5030.07 BOOL  ; DROP GUARD FORWARD
5030.08 BOOL  ; EXCHANGE CONVEYOR CW
5030.09 BOOL  ; EXCHANGE CONVEYOR CCW
5030.12 BOOL  ; PALLETIZING CONVEYOR
5030.13 BOOL  ; STACKING CONVEYOR
5040.00 BOOL  ; POSITIONING 1 BACKWARD
5040.01 BOOL  ; POSITIONING 1 FORWARD
5040.02 BOOL  ; LIFTER DOWNWARD
5040.03 BOOL  ; LIFTER UPWARD
5040.04 BOOL  ; POSITIONING 2 BACKWARD
5040.05 BOOL  ; POSITIONING 2 FORWARD
5040.06 BOOL  ; DROP GUARD BACKWARD
5040.07 BOOL  ; DROP GUARD FORWARD
5040.08 BOOL  ; EXCHANGE CONVEYOR CW
5040.09 BOOL  ; EXCHANGE CONVEYOR CCW
5040.10 BOOL  ; Writing of ID3
5040.11 BOOL  ; Writing of ID4
5040.12 BOOL  ; PALLETIZING CONVEYOR
5040.13 BOOL  ; STACKING CONVEYOR
5040.14 BOOL  ; CONVEYOR STOP
5043.00 BOOL  ; STOPPER DOWNWARD SIGNAL
5043.01 BOOL  ; Writing signal of ID3
5043.02 BOOL  ; Writing signal of ID4
5043.03 BOOL  ; STACKING CONVEYOR START SIGNAL
5043.05 BOOL  ; PALLETIZING CONVEYOR STOP SIGNAL
5043.06 BOOL  ; ﾚｰﾝ2段積み部ｺﾝﾍﾞｱ停止信号
5045.00 BOOL  ; 19ST_HOME POSITION
5045.01 BOOL  ; 19ST_CYCLE RUNNING
5052.03 BOOL  ; STACKING CONVEYOR START SIGNAL
5052.06 BOOL  ; STACKING CONVEYOR STOP SIGNAL
5052.07 BOOL  ; STACKING IMPROPRIETY
5052.08 BOOL  ; Downward confirmation when product number is switched
5052.10 BOOL  ; Disbursement completion of fraction workpiece
5053.00 BOOL  ; 20ST_1CY START PB on
5053.01 BOOL  ; 20ST_1CY RUN
5053.02 BOOL  ; 20ST_INDIV STEP START
5053.03 BOOL  ; 20ST_UNIT HOME POSITION PB
5053.04 BOOL  ; 20ST_UNIT HOME POSITION PB PLUSE
5054.00 BOOL  ; 20ST_CONDITION OF START(AUTO)
5054.01 BOOL  ; 20ST_CONDITION OF START(INDIV)
5054.04 BOOL  ; 20ST_CONDITION OF CYCLE START
5054.08 BOOL  ; 20ST_START RESET
5054.09 BOOL  ; 20ST_STEP UP ENABLE
5055.00 BOOL  ; 20ST_CYCLE RUNNING
5055.01 BOOL  ; 20ST_CYCLE RUNNING PLUSE
5055.02 BOOL  ; 20ST_STEP UP ENABLE
5055.03 BOOL  ; UNLOADING UNIT START
5055.04 BOOL  ; STACKING START
5055.05 BOOL  ; UNLOADING  START OF STACKING CONTAINER
5055.06 BOOL  ; UNLOADING PALLET CONVEYOR
5055.15 BOOL  ; 20ST_CYCLE COMPLETE
5056.08 BOOL  ; UNLOADING CONVEYOR 1
5056.12 BOOL  ; UNLOADING CONVEYOR 2
5056.13 BOOL  ; UNLOADING UNIT STOP
5057.00 BOOL  ; STACKING HOOK BACKWARD END
5057.01 BOOL  ; STACKING HOOK FORWARD END
5057.08 BOOL  ; STACKING LIFTER DOWNWARD END
5057.09 BOOL  ; STACKING LIFTER UPWARD END
5057.10 BOOL  ; STACKING LIFTER INTERMEDIATE POSITION
5080.00 BOOL  ; STACKING HOOK BACKWARD
5080.01 BOOL  ; STACKING HOOK FORWARD
5080.02 BOOL  ; STACKING LIFTER DOWNWARD
5080.03 BOOL  ; STACKING LIFTER UPWARD
5080.04 BOOL  ; STACKING CONVEYOR
5080.06 BOOL  ; STACKING STOPPER DOWNWARD
5080.07 BOOL  ; STACKING STOPPER UPWARD
5080.08 BOOL  ; UNLOADING CONVEYOR 1
5080.10 BOOL  ; UNLOADING ESCAPE UPWARD
5080.11 BOOL  ; UNLOADING ESCAPE DOWNWARD
5080.12 BOOL  ; UNLOADING CONVEYOR 2
5080.14 BOOL  ; UNLOADING STOPPER DOWNWARD
5080.15 BOOL  ; UNLOADING STOPPER UPWARD
5090.00 BOOL  ; STACKING HOOK BACKWARD
5090.01 BOOL  ; STACKING HOOK FORWARD
5090.02 BOOL  ; STACKING LIFTER DOWNWARD
5090.03 BOOL  ; STACKING LIFTER UPWARD
5090.04 BOOL  ; STACKING CONVEYOR
5090.05 BOOL  ; CONVEYOR STOP
5090.06 BOOL  ; STACKING STOPPER DOWNWARD
5090.07 BOOL  ; STACKING STOPPER UPWARD
5090.08 BOOL  ; UNLOADING CONVEYOR 1
5090.10 BOOL  ; UNLOADING ESCAPE UPWARD
5090.11 BOOL  ; UNLOADING ESCAPE DOWNWARD
5090.12 BOOL  ; UNLOADING CONVEYOR 2
5090.14 BOOL  ; UNLOADING STOPPER DOWNWARD
5090.15 BOOL  ; UNLOADING STOPPER UPWARD
5093.06 BOOL  ; STACKING CONVEYOR STOP SIGNAL
5093.07 BOOL  ; Container discharge completion
5093.08 BOOL  ; Stacking containers cannot be exchanged
5095.00 BOOL  ; 20ST_HOME POSITION
5095.01 BOOL  ; 20ST_CYCLE RUNNING
5100.00 BOOL  ; PB_Master On
5100.01 BOOL  ; PB_HOME_POS_RE
5100.02 BOOL  ; MASTER ON CONFIRM
5100.03 BOOL  ; PRO_START
5100.04 BOOL  ; HOME_POST_RE_COND
5100.05 BOOL  ; STEP_STOP_COND
5100.06 BOOL  ; MOMENT_STOP_COND
5100.07 BOOL  ; INTERRUPT_SKIP_COND
5100.08 BOOL  ; SS_PRP_INTLK
5100.09 BOOL  ; AIR_SC_CONF
5100.10 BOOL  ; SS_AUTO_IND
5100.11 BOOL  ; TEACHING ON_OFF
5100.12 BOOL  ; PL_AUTO_RUN
5100.13 BOOL  ; PB_FLT RESET
5100.14 BOOL  ; N_E_STOP
5100.15 BOOL  ; N_AUTO_STOP
5101.00 BOOL  ; STOP_COND
5101.01 BOOL  ; ENERGI_SAVING
5101.02 BOOL  ; ENERGI_SAVING_REL
5110.01 BOOL  ; EX_RB_RUNNING
5110.02 BOOL  ; EX_RB_FLT
5110.03 BOOL  ; EX_RB_SERVO_ON
5110.04 BOOL  ; EX_RB_INITIAL_COMPL
5110.05 BOOL  ; EX_RB_AUTO_MODE
5110.06 BOOL  ; EX_RB_OUTSIDE_MODE
5110.07 BOOL  ; EX_RB_BAT_WARNING
5110.08 BOOL  ; EX_RB_WARNING
5110.11 BOOL  ; EX_RB_HOME_POS
5110.14 BOOL  ; EX_COMMAND_TRTMT_COMPL
5110.15 BOOL  ; EX_RB_STATUS_ODD_PARITY
5111.00 BOOL  ; EX_RB_HOME_POS
5111.03 BOOL  ; EX_RB_MOTION_OK
5111.04 BOOL  ; EX_RB_MOTION_NG
5111.06 BOOL  ; EX_RB_SENSOR_CHK_NG
5111.07 BOOL  ; EX_RB_HAND_REP_NG
5111.08 BOOL  ; EX_RB_VISUAL NG
5130.00 BOOL  ; SIG_OFF_COMF
5130.01 BOOL  ; FLT_CODE
5130.02 BOOL  ; COMMAND_FIN
5130.03 BOOL  ; COMMAND_COMP
5130.05 BOOL  ; DATA_AREA1_BIT_EVEN
5130.06 BOOL  ; DATA_AREA2_BIT_EVEN
5130.07 BOOL  ; COMMAND_AREA_BIT_EVEN
5130.10 BOOL  ; DATA_BIT_SUM_ODD
5130.11 BOOL  ; COMMAND_TRTMT_COMPL
5130.12 BOOL  ; RB_FAULT_CLEAR_TIMING
5200.00 BOOL  ; RB_master On Condition
5200.01 BOOL  ; MSTR_ON_AIR_SC_CONF
5200.02 BOOL  ; Master On Confirm
5200.03 BOOL  ; RB_MSTR_ON_1_SCAN
5200.04 BOOL  ; MODE_CHANGE
5200.05 BOOL  ; MODE_CHANGE_COMPL
5200.06 BOOL  ; RB_HOME_POS_PB_ON
5200.07 BOOL  ; RB_HOME_POS_MOTION
5200.08 BOOL  ; RB_HOME_POS_NO_MOTION
5200.09 BOOL  ; RB_HOME_POS_COND_CONFIRM
5200.10 BOOL  ; RB_HOME_POS_PRO_START
5200.11 BOOL  ; PRO_START_RESET
5200.12 BOOL  ; RB_MSTR_ON_COMP_CLEAR_1SCAN
5200.13 BOOL  ; RB_MSTR_ON_COMP_COND
5200.14 BOOL  ; RB_MSTR_ON_COMPL
5200.15 BOOL  ; PL_RB_MSTR_ON
5201.00 BOOL  ; RB_HOME_POS_1SCAN
5201.01 BOOL  ; RB_HOME_POS_1SCAN_MEMORY
5201.02 BOOL  ; RB_HOME_POS
5201.03 BOOL  ; PL_RB_HOME_POS_RE
5201.05 BOOL  ; ENERGY_SAVING_RECEPTION
5201.06 BOOL  ; RB_PRO_START_RESET_CON
5201.07 BOOL  ; ENERGY_SAVING_REL_RECEPTION_CON
5201.09 BOOL  ; ENERGY_SAVING_REL_RECEPTION
5201.10 BOOL  ; STOP
5250.00 BOOL  ; RB_OUTSIDE_START
5250.01 BOOL  ; STROBE_SIGNAL
5250.02 BOOL  ; RB_PROSTART
5250.03 BOOL  ; RB_PRO_START_RESET
5250.04 BOOL  ; RB_RUNNING_CONFIRM
5250.05 BOOL  ; RB_MOVE_OK
5250.06 BOOL  ; RB_MOVE_NG
5400.00 BOOL  ; PL_RB_MASTER ON
5400.01 BOOL  ; PL_RB_HOME POST
5400.02 BOOL  ; CR_RB STOP
5400.03 BOOL  ; RB_FAULT
5400.04 BOOL  ; RB_BAT OFF WARNING
5400.05 BOOL  ; RB WARNING FAULT
5400.06 BOOL  ; SENSOR CHECK NG
5400.07 BOOL  ; HAND REP NG
5400.08 BOOL  ; VISION NG
5400.10 BOOL  ; RB_HOME POST
5400.11 BOOL  ; RB_MOTION OK COMPLETE
5400.12 BOOL  ; RB_MOTION NG COMPLETE
5400.13 BOOL  ; RB SERVO ON
5400.14 BOOL  ; RB_MASTER ON
5600.00 BOOL  ; Task Error Flag
5600.02 BOOL  ; Automatic Mode Flag
5600.03 BOOL  ; Manual Mode Flag
5600.04 BOOL  ; Program Execution Flag
5600.05 BOOL  ; $?St$Bk?_#[18] / Program Execution / Completed Flag$?St$Bk?_#[18]
5600.06 BOOL  ; Optional Input Standby
5600.07 BOOL  ; M Code Reset Standby
5600.08 BOOL  ; M Strobe
5600.09 BOOL  ; Cycle Start Received
5600.13 BOOL  ; Teaching Completed
5600.14 BOOL  ; Teaching Error
5600.15 BOOL  ; Teaching Address Over
5601.00 BOOL  ; Reference Origin
5601.01 BOOL  ; Busy Flag
5601.02 BOOL  ; Servo-lock ON
5601.03 BOOL  ; No Origin Flag
5601.04 BOOL  ; Axis Operating
5601.05 BOOL  ; Positioning Completed
5601.06 BOOL  ; Error Counter Warning
5601.07 BOOL  ; Alarm Input
5602.00 BOOL  ; Servo Lock
5602.01 BOOL  ; Servo Realise
5602.02 BOOL  ; Servo Origin
5604.00 BOOL  ; MC_AutoMan
5605.00 BOOL  ; Servo Motion Start Condition
5605.01 BOOL  ; Servo Motion Start
5605.02 BOOL  ; MC_Read Prog
5605.03 BOOL  ; Servo Motion Start Prog
5605.04 BOOL  ; Servo Motion Moving
5605.05 BOOL  ; Servo Motion Complete
5605.15 BOOL  ; Motion Complete
5610.00 BOOL  ; Servo Forward Position
5610.01 BOOL  ; Servo Backward Position
5650.01 BOOL  ; X AXIS TEACHING &JOG SCREEN
5650.03 BOOL  ; MASTER SWITCH ON TRIGGER
5650.04 BOOL  ; MASTER SWITCH OFF TRIGGER
5650.11 BOOL  ; X AXIS SETTING SCREEN
5651.00 BOOL  ; THE TEACHING IS ACCEPTABLE
5651.01 BOOL  ; TRANSFER ADVANCEMENT EDGE TETI COMPLETION
5651.02 BOOL  ; TRANSFER ADVANCEMENT EDGE TETI INSIDE
5651.04 BOOL  ; TRANSFER ADVANCEMENT SPEED TETI INSIDE
5651.05 BOOL  ; TRANSFER RETREAT SPEED TETI COMPLETION
5651.08 BOOL  ; FLASH MEMORY PRESERVATION TIMING
5651.09 BOOL  ; FRATSUSSHUMEMORI PRESERVATION COMPLETION
5651.10 BOOL  ; THE FLASH MEMORY IS BEING PRESERVED
5651.14 BOOL  ; TRANSFER POSITIONAL DATA READING COMPLETION
5651.15 BOOL  ; TRANSFER POSITIONAL DATA IS BEING READ
5652.00 BOOL  ; FORWARDING PERMISSION
5652.01 BOOL  ; MEMORY DRIVING END
5665.01 BOOL  ; TRANSFER ADVANCEMENT EDGE POSITION
5665.02 BOOL  ; TRANSFER ORIGINAL POSITION
5665.05 BOOL  ; TRANSFER FIXED POSITIONAL CONFIRMATION
6010.04 BOOL  ; During automatic operation from the previous process
6100 CHANNEL  ; AUTO RUNNING MACHINE
6100.01 BOOL  ; AUTO RUNNING OF MACHINE No.1
6100.02 BOOL  ; AUTO RUNNING OF MACHINE No.2
6100.03 BOOL  ; AUTO RUNNING OF MACHINE No.3
6100.04 BOOL  ; AUTO RUNNING OF MACHINE No.4
6100.05 BOOL  ; AUTO RUNNING OF MACHINE No.5
6100.06 BOOL  ; AUTO RUNNING OF MACHINE No.6
6100.07 BOOL  ; AUTO RUNNING OF MACHINE No.7
6100.08 BOOL  ; AUTO RUNNING OF MACHINE No.8
6100.09 BOOL  ; AUTO RUNNING OF MACHINE No.9
6100.10 BOOL  ; AUTO RUNNING OF MACHINE No.10
6100.11 BOOL  ; AUTO RUNNING OF MACHINE No.11
6101 CHANNEL  ; FAULT STOP MACHINE
6101.01 BOOL  ; FAULT STOP OF MACHINE No.1
6101.02 BOOL  ; FAULT STOP OF MACHINE No.2
6101.03 BOOL  ; FAULT STOP OF MACHINE No.3
6101.04 BOOL  ; FAULT STOP OF MACHINE No.4
6101.05 BOOL  ; FAULT STOP OF MACHINE No.5
6101.06 BOOL  ; FAULT STOP OF MACHINE No.6
6101.07 BOOL  ; FAULT STOP OF MACHINE No.7
6101.08 BOOL  ; FAULT STOP OF MACHINE No.8
6101.09 BOOL  ; FAULT STOP OF MACHINE No.9
6101.10 BOOL  ; FAULT STOP OF MACHINE No.10
6101.11 BOOL  ; FAULT STOP OF MACHINE No.11
6102.00 BOOL  ; ALL MACHINE OPERATING
6102.01 BOOL  ; FAULT STOP SIGNAL
6102.02 BOOL  ; DATA MEMORY
6102.03 BOOL  ; ALL MACHINE OPERATING MEMORY
6102.11 BOOL  ; PERIODICAL STOP
6102.12 BOOL  ; FAULT STOP
6102.13 BOOL  ; AUTO RUNNING STOP
6140.00 BOOL  ; CHECK BEARING NEW SENSOR
6140.01 BOOL  ; NO BEARING
6140.07 BOOL  ; KZ COLLECTING NG 291222
6142.07 BOOL  ; XXXXXX
6143.00 BOOL  ; -
6143.03 BOOL  ; Bug fix 20151125
6143.04 BOOL  ; For adjustment when there is no ID information from the previous process
6143.06 BOOL  ; Addition of finishing correction circuit
6143.07 BOOL  ; Measuring unit correction circuit
6143.09 BOOL  ; Shirai correction after 20150803
6143.10 BOOL  ; 山本修正
6143.12 BOOL  ; NO ID
6143.13 BOOL  ; Impulse measurement complete
6143.15 BOOL  ; TEMPORARY CONTACT FOR ADJUSTMENT ON
A343.13 BOOL  ; Flag when file memory operation is being executed
A343.15 BOOL  ; Memory card confirmation flag
A351 CHANNEL  ; Clock data and second
A352 CHANNEL  ; Clock data day and time
A353 CHANNEL  ; The moon clock data every year
A401.06 BOOL  ; FALS FAULT FLAG(STOP)
A402.02 BOOL  ; HIGH EFFICIENT I/O SETTING FAULT
A402.03 BOOL  ; CPU HIGH EFFICIENT I/O SETTING FAULT
A402.05 BOOL  ; SYSBUS FAULT
A402.06 BOOL  ; HIGH EFFICIENT I/O FAULT
A402.07 BOOL  ; CPU HIGH EFFICIENT I/O FAULT
A402.08 BOOL  ; INNER BOARD FAULT
A402.10 BOOL  ; FAULT IN PC SYSTEM CONSTRUCTION
A402.12 BOOL  ; FAULT IN BASIC I/O UNIT
A402.13 BOOL  ; FAULT IN INTERRUPTION TASK
A410.06 BOOL  ; High performance U of CS1 . repetition U. Number flag
A411.06 BOOL  ; High performance i/o . repetition machine Number flag
A412.04 BOOL  ; High performance i/o . repetition machine Number flag
A412.08 BOOL  ; High performance i/o . repetition machine Number flag
A417.06 BOOL  ; HIGH EFFICIENT U OF CS1 UNIT FAULT  No. FLAG
A418.06 BOOL  ; HIGH EFFICIENT I/O UNIT FAULT MACHINE No. FLAG
A419.04 BOOL  ; HIGH EFFICIENT I/O UNIT FAULT MACHINE No. FLAG
A419.08 BOOL  ; HIGH EFFICIENT I/O UNIT FAULT MACHINE No. FLAG
A427.06 BOOL  ; HIGH EFFICIENT U OF CS1 UNIT FAULT  No. FLAG
A428.06 BOOL  ; HIGH EFFICIENT I/O UNIT FAULT MACHINE No. FLAG
A429.04 BOOL  ; HIGH EFFICIENT I/O UNIT FAULT MACHINE No. FLAG
A429.08 BOOL  ; HIGH EFFICIENT I/O UNIT FAULT MACHINE No. FLAG
A502.06 BOOL  ; The sixth machine restart flag
A503.04 BOOL  ; The 20th machine restart flag
A503.08 BOOL  ; The 24th machine restart flag
C0010 BOOL  ; ID1 communication abnormality
C0011 BOOL  ; ID2 communication abnormality
C0012 BOOL  ; ID3 communication abnormality
C0013 BOOL  ; ID4 communication abnormality
C0031 BOOL  ; INSULATION TEST FAULT CONTINUALING
C0032 BOOL  ; WORK No. FAULT CONTINUALING
C0033 BOOL  ; SWING MEASUREMENT FAULT CONTINUALING
C0034 BOOL  ; RESISTANCE MEASUREMENT FAULT CONTINUALING
C0035 BOOL  ; PAIR POLE IMPULSE MEAS FAULT CONTINUALING
C0036 BOOL  ; NEXT POLE IMPULSE MEAS FAULT CONTINUALING
C0037 BOOL  ; LENGTH MEASUREMENT FAULT CONTINUALING
C0038 BOOL  ; BEARING MEASUREMENT FAULT CONTINUALING
C0043 BOOL  ; -
C0044 BOOL  ; -
C1300 BOOL  ; Repeated challenge
C1400 BOOL  ; Repeated challenge
C1450 BOOL  ; Measurement frequency (pair)
C1451 BOOL  ; Measurement frequency (next)
C1452 BOOL  ; Adjacent measurement count (for analysis)
C1454 BOOL  ; Repeated challenge
C1470 BOOL  ; Measurement frequency (pair)
C1471 BOOL  ; Measurement frequency (next)
C1500 BOOL  ; -
D0 CHANNEL  ; Screen number when being displaying it now
D100 CHANNEL  ; DATA_AREA1
D1000 CHANNEL  ; Work information received from the previous process
D10000 CHANNEL  ; QUANTITY
D10002 CHANNEL  ; DEFECTS
D10004 CHANNEL  ; INSULATION TEST DEFECTS
D10006 CHANNEL  ; SWING DEFECTS
D10008 CHANNEL  ; RESISTANCE DEFECTS
D10010 CHANNEL  ; WORKPIECE No. DEFECTS
D10012 CHANNEL  ; IMPULSE DEFECTS
D10014 CHANNEL  ; LENGTH MEASUREMENT DEFECTS (OVERALL)
D10016 CHANNEL  ; LENGTH MEASUREMENT DEFECTS (BEARING)
D10018 CHANNEL  ; LANE 1 QUANTITY
D10020 CHANNEL  ; LANE 2 QUANTITY
D10022 CHANNEL  ; RESISTANCE MEASUREMENT RETRY
D10024 CHANNEL  ; IMPULSE MEASUREMENT RETRY
D10050 CHANNEL  ; WORKPIECE No.1 QUANTITY
D10052 CHANNEL  ; WORKPIECE No.2 QUANTITY
D10054 CHANNEL  ; WORKPIECE No.3 QUANTITY
D10056 CHANNEL  ; WORKPIECE No.4 QUANTITY
D10058 CHANNEL  ; WORKPIECE No.5 QUANTITY
D1006 CHANNEL  ; Physique
D10060 CHANNEL  ; WORKPIECE No.6 QUANTITY
D10062 CHANNEL  ; WORKPIECE No.7 QUANTITY
D10064 CHANNEL  ; WORKPIECE No.8 QUANTITY
D10066 CHANNEL  ; WORKPIECE No.9 QUANTITY
D10068 CHANNEL  ; WORKPIECE No.10 QUANTITY
D10070 CHANNEL  ; WORKPIECE No.11 QUANTITY
D10072 CHANNEL  ; WORKPIECE No.12 QUANTITY
D10074 CHANNEL  ; WORKPIECE No.13 QUANTITY
D10076 CHANNEL  ; WORKPIECE No.14 QUANTITY
D10078 CHANNEL  ; WORKPIECE No.15 QUANTITY
D10080 CHANNEL  ; WORKPIECE No.16 QUANTITY
D10082 CHANNEL  ; WORKPIECE No.17 QUANTITY
D10084 CHANNEL  ; WORKPIECE No.18 QUANTITY
D10086 CHANNEL  ; WORKPIECE No.19 QUANTITY
D10088 CHANNEL  ; WORKPIECE No.20 QUANTITY
D10090 CHANNEL  ; WORKPIECE No.21 QUANTITY
D10092 CHANNEL  ; WORKPIECE No.22 QUANTITY
D10094 CHANNEL  ; WORKPIECE No.23 QUANTITY
D10096 CHANNEL  ; WORKPIECE No.24 QUANTITY
D10098 CHANNEL  ; WORKPIECE No.25 QUANTITY
D101 CHANNEL  ; DATA_AREA2_PRO_NO
D10100 CHANNEL  ; -
D10102 CHANNEL  ; INSULATION TEST ELECTRODE CHANGE PRESENT
D10104 CHANNEL  ; RESISTANCE ELECTRODE CHANGE PRESENT
D10106 CHANNEL  ; IMPULSE ELECTRODE CHANGE PRESENT
D102 CHANNEL  ; COMMAND_AREA
D10200 CHANNEL  ; QUALITY CHECK PRESENT
D10202 CHANNEL  ; INSULATION TEST ELECTRODE CHANGE NOTICE
D10204 CHANNEL  ; RESISTANCE ELECTRODE CHANGE NOTICE
D10206 CHANNEL  ; IMPULSE ELECTRODE CHANGE NOTICE
D1025 CHANNEL  ; Master Check Counting
D10300 CHANNEL  ; QUALITY CHECK STOP
D10302 CHANNEL  ; INSULATION TEST ELECTRODE CHANGE STOP
D10304 CHANNEL  ; RESISTANCE ELECTRODE CHANGE STOP
D10306 CHANNEL  ; IMPULSE ELECTRODE CHANGE STOP
D1040 CHANNEL  ; Input ST palette data storage area when forced setting Area 1
D10400 CHANNEL  ; Relay switch time
D10401 CHANNEL  ; Page set time
D10403 CHANNEL  ; Resistance measurement end time
D10404 CHANNEL  ; NUMBER OF TURNS CHECK TIMMING
D1041 CHANNEL  ; Child part number
D10418 CHANNEL  ; LUNCH TIME START
D10419 CHANNEL  ; LUNCH TIME STOP
D10420 CHANNEL  ; CYCLE TIME
D10422 CHANNEL  ; RESISTANCE MEASUREMENT RETRY
D10423 CHANNEL  ; IMPULSE MEASUREMENT RETRY
D10424 CHANNEL  ; No. SWITCH PACKING
D1046 CHANNEL  ; Physique
D1047 CHANNEL  ; Work Yes / No Information
D1048 CHANNEL  ; Processing status information
D1049 CHANNEL  ; Good / defective information
D105 CHANNEL  ; DATA_AREA1_EXTRACTION
D1050 CHANNEL  ; Input ST pallet data 1 (product number information)
D1053 CHANNEL  ; Master work No.
D1054 CHANNEL  ; Re-entry work information
D106 CHANNEL  ; DATA_AREA1_BIT_SUM
D10600 CHANNEL  ; Cycle time display
D10601 CHANNEL  ; Cycle time average display
D10620 CHANNEL  ; Cycle time count value
D107 CHANNEL  ; DATA_AREA2_BIT_SUM
D10704 CHANNEL  ; OPERATION RATE
D108 CHANNEL  ; COMMAND_AREA_BIT_SUM
D1080 CHANNEL  ; Input ST palette data storage area 2 (independent operation mode) when forced setting
D10800 CHANNEL  ; QUANTITY   X   CYCLE TIME
D10810 CHANNEL  ; QUANTITY   X   CYCLE TIME   X   100
D10820 CHANNEL  ; QUANTITY   X   CYCLE TIME   X   100
D10830 CHANNEL  ; QUANTITY   X   CYCLE TIME   /   100
D1086 CHANNEL  ; Physique
D1087 CHANNEL  ; Work Yes / No Information
D1088 CHANNEL  ; Processing status information
D1089 CHANNEL  ; Good / defective information
D1090 CHANNEL  ; Work completion information
D10900 CHANNEL  ; RESISTANCE 1 PAIR POLE NG
D10902 CHANNEL  ; RESISTANCE 2 PAIR POLE NG
D10904 CHANNEL  ; RESISTANCE 3 PAIR POLE NG
D10906 CHANNEL  ; RESISTANCE 4 PAIR POLE NG
D10908 CHANNEL  ; RESISTANCE 5 PAIR POLE NG
D10910 CHANNEL  ; RESISTANCE 6 PAIR POLE NG
D10912 CHANNEL  ; RESISTANCE 7 80 NG
D10914 CHANNEL  ; RESISTANCE 8 80 NG
D10916 CHANNEL  ; RESISTANCE 9 80 NG
D10924 CHANNEL  ; RESISTANCE 1 180 NG
D10926 CHANNEL  ; RESISTANCE 2 180 NG
D10928 CHANNEL  ; RESISTANCE 3 180 NG
D10930 CHANNEL  ; RESISTANCE 4 180 NG
D10932 CHANNEL  ; RESISTANCE 5 180 NG
D10934 CHANNEL  ; RESISTANCE 6 180 NG
D10936 CHANNEL  ; RESISTANCE 7 180 NG
D10938 CHANNEL  ; RESISTANCE 8 180 NG
D10940 CHANNEL  ; RESISTANCE 9 180 NG
D120 CHANNEL  ; ROBOT PROG MEMORY
D122 CHANNEL  ; WORD: RB_FAULT
D1282 CHANNEL  ; OPERATIONTIME
D1300 CHANNEL  ; POINT SETTING SMALL NUMBER OF FORWARD SPEEDS
D1301 CHANNEL  ; ADVANCEMENT POSITION SETTING PLC
D1303 CHANNEL  ; POINT SETTING OF SMALL NUMBER OF ADVANCEMENT EDGES
D1306 CHANNEL  ; POINT SETTING OF SMALL NUMBER OF RETREAT SPEEDS
D1309 CHANNEL  ; RETREAT POSITION DECIMAL POINT SETTING
D1310 CHANNEL  ; RETREAT POSITION SETTING PLC
D1312 CHANNEL  ; PRELIMINARY DECIMAL POINT SETTING
D1350 CHANNEL  ; WORKPIECE TEMPERATURE READ(BCD)
D1400 CHANNEL  ; JOG SPEED %
D1410 CHANNEL  ; ROBOT PROGRAM NUMBER SET
D1510 CHANNEL  ; FLASH MEMORY PRESERVATION COMMAND
D16 CHANNEL  ; FOR FAULT WINDOW INDICATION
D17 CHANNEL  ; FAULT WINDOW NUMBER SETUP
D1700 CHANNEL  ; CODE No. OFFSET
D1701 CHANNEL  ; CODE No. OFFSET
D1750 CHANNEL  ; CODE No. OFFSET
D1751 CHANNEL  ; CODE No. OFFSET
D1769 CHANNEL  ; IMPULSE NEXT POLE PAGE No.
D18 CHANNEL  ; FAULT WINDOW X COORDINATES
D1800 CHANNEL  ; PAIR POLE MEASUREMENT NUMBER OF TIMES
D1803 CHANNEL  ; IMPULSE PAIR POLE EXCITATION PATTERN DM STORING
D1804 CHANNEL  ; Impulse anti-polar excitation pattern storage
D1806 CHANNEL  ; IMPULSE PAIR POLE EXCITATION PATTERN DM STORING(INDIVIDUAL)
D1808 CHANNEL  ; IMPULSE PAIR POLE PAGE No. (BIN)
D1809 CHANNEL  ; IMPULSE PAIR POLE PROGRAM No. (BIN)
D1810 CHANNEL  ; NEXT POLE MEASUREMENT NUMBER OF TIMES
D1813 CHANNEL  ; IMPULSE NEXT POLE EXCITATION PATTERN DM STORING
D1814 CHANNEL  ; Impulse adjacent excitation pattern storage
D1816 CHANNEL  ; IMPULSE NEXT POLE EXCITATION PATTERN DM STORING(INDIVIDUAL)
D1818 CHANNEL  ; IMPULSE NEXT POLE PAGE No. (BIN)
D1819 CHANNEL  ; IMPULSE NEXT POLE PROGRAM No.(BIN)
D19 CHANNEL  ; FAULT WINDOW Y COORDINATES
D2 CHANNEL  ; 年現在値 (ﾀｯﾁﾊﾟﾈﾙより)
D2000 CHANNEL  ; Priset value of high-speed counter
D2002 CHANNEL  ; Count value of high-speed counter
D2004 CHANNEL  ; LENGTH MEASUREMENT DATA (OVERALL)
D2010 CHANNEL  ; Priset value of high-speed counter
D2012 CHANNEL  ; Count value of high-speed counter
D2014 CHANNEL  ; LENGTH MEASUREMENT DATA (BEARING)
D20600 CHANNEL  ; AD041 USE SPECIFICATION
D20601 CHANNEL  ; AD041 RANGE SPECIFICATION
D20602 CHANNEL  ; AD041 INPUT 1 EQUALIZATION PROCESSING
D20620 CHANNEL  ; OFFSET
D20621 CHANNEL  ; SCALING X VALUE
D20622 CHANNEL  ; SCALING Y VALUE
D2111 CHANNEL  ; Memory of packing in a container of fraction workpiece (code no.1)
D2112 CHANNEL  ; Memory of packing in a container of fraction workpiece (code no.2)
D2113 CHANNEL  ; Memory of packing in a container of fraction workpiece (code no.3)
D2114 CHANNEL  ; Memory of packing in a container of fraction workpiece (code no.4)
D2115 CHANNEL  ; Memory of packing in a container of fraction workpiece (code no.5)
D2116 CHANNEL  ; Memory of packing in a container of fraction workpiece (code no.6)
D2117 CHANNEL  ; Memory of packing in a container of fraction workpiece (code no.7)
D2118 CHANNEL  ; Memory of packing in a container of fraction workpiece (code no.8)
D2119 CHANNEL  ; Memory of packing in a container of fraction workpiece (code no.9)
D2121 CHANNEL  ; Number of packing in a container of fraction workpiece (code no.1)
D2122 CHANNEL  ; Number of packing in a container of fraction workpiece (code no.2)
D2123 CHANNEL  ; Number of packing in a container of fraction workpiece (code no.3)
D2124 CHANNEL  ; Number of packing in a container of fraction workpiece (code no.4)
D2125 CHANNEL  ; Number of packing in a container of fraction workpiece (code no.5)
D2126 CHANNEL  ; Number of packing in a container of fraction workpiece (code no.6)
D2127 CHANNEL  ; Number of packing in a container of fraction workpiece (code no.7)
D2128 CHANNEL  ; Number of packing in a container of fraction workpiece (code no.8)
D2129 CHANNEL  ; Number of packing in a container of fraction workpiece (code no.9)
D213 CHANNEL  ; LANE 1 WORKPIECE NUMBER DISPLAY
D2131 CHANNEL  ; The following position of packing in a container number in fraction workpiece (code no.1)
D2132 CHANNEL  ; The following position of packing in a container number in fraction workpiece (code no.2)
D2133 CHANNEL  ; The following position of packing in a container number in fraction workpiece (code no.3)
D2134 CHANNEL  ; The following position of packing in a container number in fraction workpiece (code no.4)
D2135 CHANNEL  ; The following position of packing in a container number in fraction workpiece (code no.5)
D2136 CHANNEL  ; The following position of packing in a container number in fraction workpiece (code no.6)
D2137 CHANNEL  ; The following position of packing in a container number in fraction workpiece (code no.7)
D2138 CHANNEL  ; The following position of packing in a container number in fraction workpiece (code no.8)
D2139 CHANNEL  ; The following position of packing in a container number in fraction workpiece (code no.9)
D214 CHANNEL  ; LANE 2 WORKPIECE NUMBER DISPLAY
D2141 CHANNEL  ; The following position of taking out in a container number in fraction workpiece (code no.1)
D2142 CHANNEL  ; The following position of taking out in a container number in fraction workpiece (code no.2)
D2143 CHANNEL  ; The following position of taking out in a container number in fraction workpiece (code no.3)
D2144 CHANNEL  ; The following position of taking out in a container number in fraction workpiece (code no.4)
D2145 CHANNEL  ; The following position of taking out in a container number in fraction workpiece (code no.5)
D2146 CHANNEL  ; The following position of taking out in a container number in fraction workpiece (code no.6)
D2147 CHANNEL  ; The following position of taking out in a container number in fraction workpiece (code no.7)
D2148 CHANNEL  ; The following position of taking out in a container number in fraction workpiece (code no.8)
D2149 CHANNEL  ; The following position of taking out in a container number in fraction workpiece (code no.9)
D215 CHANNEL  ; LANE 1 WORKPIECE NUMBER
D2150 CHANNEL  ; Taking out positional number in fraction workpiece
D216 CHANNEL  ; LANE 2 WORKPIECE NUMBER
D2161 CHANNEL  ; Number of packing in a container of lane 1 (exchange container)(BIN)
D2162 CHANNEL  ; Number of packing in a container of lane 2 (exchange container)(BIN)
D2163 CHANNEL  ; Number of packing in a container of lane 1 (container before exchange)(BIN)
D2164 CHANNEL  ; Number of packing in a container of lane 2 (container before exchange)(BIN)
D217 CHANNEL  ; LANE 1 WORKPIECE PRODUCT NUMBER
D2171 CHANNEL  ; Next position of packing in a container of lane 1 (exchange container)(BIN)
D2172 CHANNEL  ; Next position of packing in a container of lane 2 (exchange container)(BIN)
D2173 CHANNEL  ; Next position of packing in a container of lane 3 (exchange container)(BIN)
D2174 CHANNEL  ; Next position of packing in a container of lane 4 (exchange container)(BIN)
D218 CHANNEL  ; LANE 2 WORKPIECE PRODUCT NUMBER
D2180 CHANNEL  ; Unloading position number
D2182 CHANNEL  ; Container exhaust position number in fraction workpiece
D219 CHANNEL  ; LANE 2 WORKPIECE NEXT PRODUCT NUMBER
D2191 CHANNEL  ; LANE 1 WORKPIECE PRODUCT NUMBER
D2192 CHANNEL  ; LANE 2 WORKPIECE PRODUCT NUMBER
D220 CHANNEL  ; CODE No.(SCREEN)
D2200 CHANNEL  ; Movement position number
D22030 CHANNEL  ; Mode setting of counter 1
D22031 CHANNEL  ; Setting of twice counter 1
D2208 CHANNEL  ; Number of bearing taking out
D221 CHANNEL  ; PARENTS WORKPIECE NUMBER(SCREEN)
D2210 CHANNEL  ; Taking out position
D22120 CHANNEL  ; Mode setting of counter 3
D22121 CHANNEL  ; Setting of twice counter 3
D22430 CHANNEL  ; Mode setting of counter 1
D22431 CHANNEL  ; Setting of twice counter 1
D225 CHANNEL  ; PAIR POLE RESISTANCE SPECIFICATION MINIMUM VALUE(SCREEN)
D22520 CHANNEL  ; Mode setting of counter 3
D22521 CHANNEL  ; Setting of twice counter 3
D246 CHANNEL  ; SET DATA (THICKNESS OF CORE)
D247 CHANNEL  ; SET DATA (COIL END)
D248 CHANNEL  ; SET DATA (BEARING INSERT)
D250 CHANNEL  ; Swinging width standard value (worm)
D252 CHANNEL  ; Swinging width standard value (shaft end)
D3 CHANNEL  ; GP MONTH
D300 CHANNEL  ; Resistance counter electrode data 9 (80 ° counter electrode)
D30000 CHANNEL  ; DATA LINK PARAMETER AREA N
D30001 CHANNEL  ; DATA LINK PARAMETER AREA N+1
D30002 CHANNEL  ; DATA LINK PARAMETER AREA N+2
D30003 CHANNEL  ; DATA LINK PARAMETER AREA N+3
D30004 CHANNEL  ; DATA LINK PARAMETER AREA N+4
D30005 CHANNEL  ; DATA LINK PARAMETER AREA N+5
D30006 CHANNEL  ; DATA LINK PARAMETER AREA N+6
D30007 CHANNEL  ; DATA LINK PARAMETER AREA N+7
D30008 CHANNEL  ; DATA LINK PARAMETER AREA N+8
D30009 CHANNEL  ; DATA LINK PARAMETER AREA N+9
D30011 CHANNEL  ; DATA LINK PARAMETER AREA N+11
D305 CHANNEL  ; PAIR POLE RESISTANCE MEASUREMENT DATA 6
D308 CHANNEL  ; Resistance counter electrode data 1 (80 ° counter electrode)
D329 CHANNEL  ; PAIR POLE RESISTANCE DATA INDIRECT SPECIFICATION
D330 CHANNEL  ; Resistance counter electrode data 1 (180 ° counter electrode)
D338 CHANNEL  ; Resistor counter electrode data 9 (180 ° counter electrode)
D3500 CHANNEL  ; Quantity of 8:40 9:40
D3501 CHANNEL  ; Quantity of 9:40 10:40
D3502 CHANNEL  ; Quantity of 10:40 11:40
D3503 CHANNEL  ; Quantity of 11:40 13:40
D3504 CHANNEL  ; Quantity of 13:25 14:25
D3505 CHANNEL  ; Quantity of 14:25 15:25
D3506 CHANNEL  ; Quantity of 15:25 16:25
D3507 CHANNEL  ; Quantity of 16:25 17:15
D3508 CHANNEL  ; Quantity of 17:15 18:30
D3509 CHANNEL  ; Quantity of 18:30 19:30
D3510 CHANNEL  ; Quantity of 19:30 19:55
D3520 CHANNEL  ; Quantity of each every time
D3530 CHANNEL  ; Time
D359 CHANNEL  ; Indirect designation of resistance counter electrode data (180 °)
D3600 CHANNEL  ; Operation time (For operation rate)
D370 CHANNEL  ; NUMBER OF TIMES SET VALUE OF RESISTANCE MEASUREMENT
D3700 CHANNEL  ; Quantity (For operation rate)
D371 CHANNEL  ; NUMBER OF TIMES OF PAIR POLE RESISTANCE PRESENT MEASUREMENT
D372 CHANNEL  ; Counter electrode resistance measurement indirect (80 °)
D373 CHANNEL  ; Counter electrode resistance measurement indirect (80 °)
D374 CHANNEL  ; 180°対極抵抗測定回数設定値
D375 CHANNEL  ; Counter electrode resistance Current measurement count (180 °)
D376 CHANNEL  ; Counter electrode resistance Current measurement count (180 °)
D377 CHANNEL  ; RESISTANCE　OFFSET
D380 CHANNEL  ; RESISTANCE READING VALUE LOW DIGIT
D381 CHANNEL  ; RESISTANCE READING VALUE HIGH DIGIT
D382 CHANNEL  ; FOR OPERATION
D384 CHANNEL  ; FOR OPERATION
D386 CHANNEL  ; FOR OPERATION
D390 CHANNEL  ; WORKPIECE TEMPERATURE READING(BCD)
D391 CHANNEL  ; WORKPIECE TEMPERATURE(BCD) HIGH DIGIT
D392 CHANNEL  ; TEMPERATURE COEFFICIENT SET VALUE
D394 CHANNEL  ; TEMPERATURE CORRECTION OPERATION LOW DIGIT
D396 CHANNEL  ; EFFECTIVE 4 DIGIT AS RESULT OF TEMPERATURE CORRECTION
D4 CHANNEL  ; GP DAY
D40 CHANNEL  ; FAULT NUMBER OF INDICATION
D41 CHANNEL  ; FAULT NUMBER WITH LAST SCAN
D410 CHANNEL  ; Swinging measurements (shaft end)
D4100 CHANNEL  ; IMPULSE NEXT POLE EXCITATION PATTERN 1-2
D4101 CHANNEL  ; IMPULSE NEXT POLE EXCITATION PATTERN 2-3
D4102 CHANNEL  ; IMPULSE NEXT POLE EXCITATION PATTERN 3-4
D4103 CHANNEL  ; IMPULSE NEXT POLE EXCITATION PATTERN 4-5
D4104 CHANNEL  ; IMPULSE NEXT POLE EXCITATION PATTERN 5-6
D4105 CHANNEL  ; IMPULSE NEXT POLE EXCITATION PATTERN 6-7
D4106 CHANNEL  ; IMPULSE NEXT POLE EXCITATION PATTERN 7-8
D4107 CHANNEL  ; IMPULSE NEXT POLE EXCITATION PATTERN 8-9
D4108 CHANNEL  ; IMPULSE NEXT POLE EXCITATION PATTERN 9-10
D4109 CHANNEL  ; IMPULSE NEXT POLE EXCITATION PATTERN 10-11
D4110 CHANNEL  ; IMPULSE NEXT POLE EXCITATION PATTERN 10-12
D4111 CHANNEL  ; IMPULSE NEXT POLE EXCITATION PATTERN 12-1
D414 CHANNEL  ; Swinging measurements (worm)
D415 CHANNEL  ; Swinging judgment (sshaft end)
D4160 CHANNEL  ; IMPULSE PAIR POLE EXCITATION PATTERN 1-7
D4161 CHANNEL  ; IMPULSE PAIR POLE EXCITATION PATTERN 2-8
D4162 CHANNEL  ; IMPULSE PAIR POLE EXCITATION PATTERN 3-9
D4163 CHANNEL  ; IMPULSE PAIR POLE EXCITATION PATTERN 4-10
D4164 CHANNEL  ; IMPULSE PAIR POLE EXCITATION PATTERN 5-11
D4165 CHANNEL  ; IMPULSE PAIR POLE EXCITATION PATTERN 6-12
D4190 CHANNEL  ; IMPULSE PAIR POLE EXCITATION PATTERN 1-5
D4191 CHANNEL  ; IMPULSE PAIR POLE EXCITATION PATTERN 2-6
D4192 CHANNEL  ; IMPULSE PAIR POLE EXCITATION PATTERN 3-7
D4193 CHANNEL  ; IMPULSE PAIR POLE EXCITATION PATTERN 4-8
D4194 CHANNEL  ; IMPULSE PAIR POLE EXCITATION PATTERN 5-9
D4195 CHANNEL  ; IMPULSE PAIR POLE EXCITATION PATTERN 6-10
D4196 CHANNEL  ; IMPULSE PAIR POLE EXCITATION PATTERN 7-11
D4197 CHANNEL  ; IMPULSE PAIR POLE EXCITATION PATTERN 8-12
D4198 CHANNEL  ; IMPULSE PAIR POLE EXCITATION PATTERN 9-13
D4199 CHANNEL  ; IMPULSE PAIR POLE EXCITATION PATTERN 10-14
D42 CHANNEL  ; FAULT CH SEARCH CONTROL VALUE
D420 CHANNEL  ; The previous swinging measurements (shaft end)
D4200 CHANNEL  ; IMPULSE PAIR POLE EXCITATION PATTERN 11-15
D4201 CHANNEL  ; IMPULSE PAIR POLE EXCITATION PATTERN 12-16
D4202 CHANNEL  ; IMPULSE PAIR POLE EXCITATION PATTERN 13-17
D4203 CHANNEL  ; IMPULSE PAIR POLE EXCITATION PATTERN 14-18
D4204 CHANNEL  ; IMPULSE PAIR POLE EXCITATION PATTERN 15-1
D4205 CHANNEL  ; IMPULSE PAIR POLE EXCITATION PATTERN 16-2
D4206 CHANNEL  ; IMPULSE PAIR POLE EXCITATION PATTERN 17-3
D4207 CHANNEL  ; IMPULSE PAIR POLE EXCITATION PATTERN 18-1
D422 CHANNEL  ; Maximum of swinging (shaft end)
D4220 CHANNEL  ; RESISTANCE PAIR POLE EXCITATION PATTERN 1-7
D4221 CHANNEL  ; RESISTANCE PAIR POLE EXCITATION PATTERN 2-8
D4222 CHANNEL  ; RESISTANCE PAIR POLE EXCITATION PATTERN 3-9
D4223 CHANNEL  ; RESISTANCE PAIR POLE EXCITATION PATTERN 4-10
D4224 CHANNEL  ; RESISTANCE PAIR POLE EXCITATION PATTERN 5-11
D4225 CHANNEL  ; RESISTANCE PAIR POLE EXCITATION PATTERN 6-12
D4226 CHANNEL  ; RESISTANCE PAIR POLE EXCITATION PATTERN 7-11
D424 CHANNEL  ; Minimum of swinging (shaft end)
D4250 CHANNEL  ; RESISTANCE PAIR POLE EXCITATION PATTERN 1-5
D4251 CHANNEL  ; RESISTANCE PAIR POLE EXCITATION PATTERN 2-6
D4252 CHANNEL  ; RESISTANCE PAIR POLE EXCITATION PATTERN 3-7
D4253 CHANNEL  ; RESISTANCE PAIR POLE EXCITATION PATTERN 4-8
D4254 CHANNEL  ; RESISTANCE PAIR POLE EXCITATION PATTERN 5-9
D4255 CHANNEL  ; RESISTANCE PAIR POLE EXCITATION PATTERN 6-10
D4256 CHANNEL  ; RESISTANCE PAIR POLE EXCITATION PATTERN 7-11
D4257 CHANNEL  ; RESISTANCE PAIR POLE EXCITATION PATTERN 8-12
D4258 CHANNEL  ; RESISTANCE PAIR POLE EXCITATION PATTERN 9-13
D426 CHANNEL  ; Swinging measurement result (shaft end)
D427 CHANNEL  ; Swinging measurement result (shaft end)
D43 CHANNEL  ; FAULT BIT NUMBER(BCD)
D430 CHANNEL  ; The previous swinging measurements (worm)
D432 CHANNEL  ; Maximum of swinging (worm)
D434 CHANNEL  ; Minimum of swinging (worm)
D436 CHANNEL  ; Swinging measurement result (worm)
D437 CHANNEL  ; Swinging measurement result (worm)
D44 CHANNEL  ; RESET BIT CONTROL VALUE
D4400 CHANNEL  ; STORED RESISTANCE
D4402 CHANNEL  ; RESISTANCE MEASURED VALUE
D4403 CHANNEL  ; RESISTANCE MEASURED VALUE UPPER 3 DIGITS
D4404 CHANNEL  ; RESISTANCE MEASURED VALUE(TEMPORARILY SAVED)
D4410 CHANNEL  ; TEMPERATURE ADJUST FOR CALCULATION(BCD LOWER 4 DIGITS)
D4412 CHANNEL  ; TEMPERATURE COEFFICIENT SET VALUE(BCD LOWER 4 DIGITS)
D4414 CHANNEL  ; FOR CALCULATION
D4418 CHANNEL  ; FOR TEMPERATURE ADJUST DENOMINATOR VALUE(BCD LOWER 4 DIGITS)
D4420 CHANNEL  ; RESISTANCE VALUE *10(BCD LOWER 4 DIGITS)
D4424 CHANNEL  ; ADJUST RESISTANCE VALUE AFTER TEMPERATURE CALCULATION RESULT QUOTIENT(BCD LOWER 4 DIGITS)
D4443 CHANNEL  ; ADJUST RESISTANCE VALUE AFTER TEMPERATURE CALCULATION RESULT QUOTIENT(BCD UPPER 4 DIGITS)
D4451 CHANNEL  ; ADJUST RESISTANCE VALUE AFTER TEMPERATURE POSITIVE NUMBER 2 DIGITS(BCD 2 DIGITS)
D5 CHANNEL  ; GP HOUR&MINUTE
D50 CHANNEL  ; FOR MONITOR INDICATION
D5000 CHANNEL  ; Results of 7:55 8:40
D5002 CHANNEL  ; Results of 8:40 9:40
D5004 CHANNEL  ; Results of 9:40 10:40
D5006 CHANNEL  ; Results of 10:40 11:40
D5008 CHANNEL  ; Results of 11:40 13:25
D5010 CHANNEL  ; Results of 13:25 14:25
D5012 CHANNEL  ; Results of 14:25 15:25
D5014 CHANNEL  ; Results of 15:25 16:25
D5016 CHANNEL  ; Results of 16:25 17:15
D5018 CHANNEL  ; Results of 17:15 18:30
D5020 CHANNEL  ; Results of 18:30 19:30
D5022 CHANNEL  ; Results of 19:30 19:55
D5030 CHANNEL  ; Accumulation of 7:55 8:40
D5032 CHANNEL  ; Accumulation of 8:40 9:40
D5034 CHANNEL  ; Accumulation of 9:40 10:40
D5036 CHANNEL  ; Accumulation of 10:40 11:40
D5038 CHANNEL  ; Accumulation of 11:40 13:25
D5040 CHANNEL  ; Accumulation of 13:25 14:25
D5042 CHANNEL  ; Accumulation of 14:25 15:25
D5044 CHANNEL  ; Accumulation of 15:25 16:25
D5046 CHANNEL  ; Accumulation of 16:25 17:15
D5048 CHANNEL  ; Accumulation of 17:15 18:30
D5050 CHANNEL  ; Accumulation of 18:30 19:30
D5052 CHANNEL  ; Accumulation of 19:30 19:55
D5060 CHANNEL  ; Operation rate of 8:40 9:40
D5062 CHANNEL  ; Operation rate of 9:40 10:40
D5064 CHANNEL  ; Operation rate of 10:40 11:40
D5066 CHANNEL  ; Operation rate of 11:40 13:25
D5068 CHANNEL  ; Operation rate of 13:25 14:25
D5070 CHANNEL  ; Operation rate of 14:25 15:25
D5072 CHANNEL  ; Operation rate of 15:25 16:25
D5074 CHANNEL  ; Operation rate of 16:25 17:15
D5076 CHANNEL  ; Operation rate of 17:15 18:30
D5078 CHANNEL  ; Operation rate of 18:30 19:30
D5080 CHANNEL  ; Operation rate of 19:30 19:55
D5090 CHANNEL  ; QUANTITY
D51 CHANNEL  ; FOR MONITOR NUMBER SETUP
D52 CHANNEL  ; MONITOR INDICATION X COORDINATES
D520 CHANNEL  ; Abnormal code storage area
D53 CHANNEL  ; MONITOR INDICATION Y COORDINATES
D55 CHANNEL  ; USED KEYBOARD NUMBER SETUP
D550 CHANNEL  ; Master work type No.
D56 CHANNEL  ; X COORDINATES
D560 CHANNEL  ; Number of master work imports
D57 CHANNEL  ; Y COORDINATES
D60 CHANNEL  ; FOR WINDOW INDICATION AT INDIVIDUAL
D6000 CHANNEL  ; 時間稼働率計算用
D6010 CHANNEL  ; For calculation
D6020 CHANNEL  ; For calculation
D6030 CHANNEL  ; Time operationrate
D6040 CHANNEL  ; For calculation
D61 CHANNEL  ; CHARACTER TABLE SETUP
D63 CHANNEL  ; USED KEYBOARD NUMBER SETUP
D64 CHANNEL  ; X COORDINATES
D65 CHANNEL  ; Y COORDINATES
D66 CHANNEL  ; FOR SET CONFIRMATION DISPLAY
D67 CHANNEL  ; SET CONFIRMATION NO.
D68 CHANNEL  ; SET CONFIRMATION DISPLAY POSITION
D70 CHANNEL  ; FAULT CH STORING HEAD DM
D7000 CHANNEL  ; -
D7001 CHANNEL  ; -
D7002 CHANNEL  ; -
D7003 CHANNEL  ; -
D7004 CHANNEL  ; -
D7005 CHANNEL  ; -
D7006 CHANNEL  ; -
D7007 CHANNEL  ; -
D7008 CHANNEL  ; -
D7009 CHANNEL  ; -
D7010 CHANNEL  ; -
D7011 CHANNEL  ; -
D7012 CHANNEL  ; -
D7013 CHANNEL  ; -
D7014 CHANNEL  ; -
D7015 CHANNEL  ; -
D7016 CHANNEL  ; -
D7017 CHANNEL  ; -
D7018 CHANNEL  ; -
D7019 CHANNEL  ; -
D7020 CHANNEL  ; -
D7021 CHANNEL  ; -
D7022 CHANNEL  ; -
D7023 CHANNEL  ; -
D7024 CHANNEL  ; -
D7025 CHANNEL  ; -
D7026 CHANNEL  ; -
D7027 CHANNEL  ; -
D7028 CHANNEL  ; -
D7029 CHANNEL  ; -
D7030 CHANNEL  ; -
D7031 CHANNEL  ; -
D7032 CHANNEL  ; -
D7033 CHANNEL  ; -
D7034 CHANNEL  ; -
D7035 CHANNEL  ; -
D7036 CHANNEL  ; -
D7037 CHANNEL  ; -
D7038 CHANNEL  ; -
D7039 CHANNEL  ; -
D7040 CHANNEL  ; -
D7041 CHANNEL  ; -
D7042 CHANNEL  ; -
D7043 CHANNEL  ; -
D7044 CHANNEL  ; -
D7045 CHANNEL  ; -
D7046 CHANNEL  ; -
D7047 CHANNEL  ; -
D7048 CHANNEL  ; -
D7049 CHANNEL  ; -
D7050 CHANNEL  ; -
D7051 CHANNEL  ; -
D7052 CHANNEL  ; -
D7100 CHANNEL  ; -
D7300 CHANNEL  ; -
D7306 CHANNEL  ; -
D7312 CHANNEL  ; -
D7318 CHANNEL  ; -
D7324 CHANNEL  ; -
D7330 CHANNEL  ; -
D7336 CHANNEL  ; -
D7342 CHANNEL  ; -
D7348 CHANNEL  ; -
D7354 CHANNEL  ; -
D7360 CHANNEL  ; -
D7366 CHANNEL  ; -
D7372 CHANNEL  ; -
D7378 CHANNEL  ; -
D7384 CHANNEL  ; -
D7390 CHANNEL  ; -
D7396 CHANNEL  ; -
D7402 CHANNEL  ; -
D7408 CHANNEL  ; -
D7414 CHANNEL  ; -
D7420 CHANNEL  ; -
D7426 CHANNEL  ; -
D7432 CHANNEL  ; -
D7438 CHANNEL  ; -
D7444 CHANNEL  ; -
D7450 CHANNEL  ; -
D7456 CHANNEL  ; -
D7461 CHANNEL  ; -
D7500 CHANNEL  ; -
D7502 CHANNEL  ; -
D7504 CHANNEL  ; -
D7506 CHANNEL  ; -
D7508 CHANNEL  ; -
D7510 CHANNEL  ; -
D7512 CHANNEL  ; -
D7514 CHANNEL  ; -
D7516 CHANNEL  ; -
D7518 CHANNEL  ; -
D7520 CHANNEL  ; -
D7522 CHANNEL  ; -
D7524 CHANNEL  ; -
D7526 CHANNEL  ; -
D7528 CHANNEL  ; -
D7530 CHANNEL  ; -
D7532 CHANNEL  ; -
D7534 CHANNEL  ; -
D7536 CHANNEL  ; -
D7538 CHANNEL  ; -
D7540 CHANNEL  ; -
D7542 CHANNEL  ; -
D7544 CHANNEL  ; -
D7546 CHANNEL  ; -
D7548 CHANNEL  ; -
D7550 CHANNEL  ; -
D7552 CHANNEL  ; -
D7553 CHANNEL  ; -
D7600 CHANNEL  ; -
D7700 CHANNEL  ; -
D7800 CHANNEL  ; -
D7907 CHANNEL  ; -
D7960 CHANNEL  ; -
D7961 CHANNEL  ; -
D7962 CHANNEL  ; -
D7963 CHANNEL  ; -
D7964 CHANNEL  ; -
D8 CHANNEL  ; CHANGE SCREEN NUMBER
D800 CHANNEL  ; Reference address storage
D802 CHANNEL  ; Reading head address set
D804 CHANNEL  ; The start address is temporarily memorized
D806 CHANNEL  ; The data storage head address is memorized
D808 CHANNEL  ; Reading byte number set
D810 CHANNEL  ; ID1 WORKPIECE NUMBER
D816 CHANNEL  ; Number of packing in a containrt(BCD)
D817 CHANNEL  ; WORKPIECE NUMBER (BCD)
D824 CHANNEL  ; The start address is temporarily memorized
D826 CHANNEL  ; The data storage head address is memorized
D828 CHANNEL  ; Writing number of words
D830 CHANNEL  ; Writing workpiece number data
D831 CHANNEL  ; Writing equipment number data
D832 CHANNEL  ; The moon on writing clock data day
D833 CHANNEL  ; Amount at writing clock data
D836 CHANNEL  ; Number of packing in a containrt(BCD)
D837 CHANNEL  ; One lane flow workpiece number
D840 CHANNEL  ; Number of packing in a containrt(BIN)
D842 CHANNEL  ; Control data
D844 CHANNEL  ; Forwarding data
D850 CHANNEL  ; Reference address storage
D852 CHANNEL  ; Reading head address set
D854 CHANNEL  ; The start address is temporarily memorized
D856 CHANNEL  ; The data storage head address is memorized
D858 CHANNEL  ; Reading byte number set
D860 CHANNEL  ; ID2 WORKPIECE NUMBER
D866 CHANNEL  ; Number of packing in a containrt(BCD)
D867 CHANNEL  ; WORKPIECE NUMBER (BCD)
D874 CHANNEL  ; The start address is temporarily memorized
D876 CHANNEL  ; The data storage head address is memorized
D878 CHANNEL  ; Writing number of words
D880 CHANNEL  ; Writing workpiece number data
D881 CHANNEL  ; Writing equipment number data
D882 CHANNEL  ; The moon on writing clock data day
D883 CHANNEL  ; Amount at writing clock data
D886 CHANNEL  ; Number of packing in a containrt(BCD)
D887 CHANNEL  ; One lane flow workpiece number
D890 CHANNEL  ; Number of packing in a containrt(BIN)
D892 CHANNEL  ; Control data
D894 CHANNEL  ; Forwarding data
D900 CHANNEL  ; Reference address storage
D902 CHANNEL  ; Reading head address set
D904 CHANNEL  ; The start address is temporarily memorized
D906 CHANNEL  ; The data storage head address is memorized
D908 CHANNEL  ; Reading byte number set
D910 CHANNEL  ; ID3 WORKPIECE NUMBER
D916 CHANNEL  ; Number of packing in a containrt(BCD)
D917 CHANNEL  ; WORKPIECE NUMBER (BCD)
D924 CHANNEL  ; The start address is temporarily memorized
D926 CHANNEL  ; The data storage head address is memorized
D9260 CHANNEL  ; CODE No. MEMORY
D9261 CHANNEL  ; CODE No. OFFSET
D9262 CHANNEL  ; CODE No. OFFSET
D9263 CHANNEL  ; SPECIFICATION VALUE ADDRESS INDIRECT SPECIFICATION
D9264 CHANNEL  ; SPECIFICATION VALUE MEMORY
D928 CHANNEL  ; Writing number of words
D9280 CHANNEL  ; SPECIFICATION VALUE ADDRESS INDIRECT SPECIFICATION
D930 CHANNEL  ; Writing workpiece number data
D931 CHANNEL  ; Writing equipment number data
D932 CHANNEL  ; The moon on writing clock data day
D933 CHANNEL  ; Amount at writing clock data
D936 CHANNEL  ; Number of packing in a containrt(BCD)
D937 CHANNEL  ; One lane flow workpiece number
D940 CHANNEL  ; Number of packing in a containrt(BIN)
D942 CHANNEL  ; Control data
D944 CHANNEL  ; Forwarding data
D950 CHANNEL  ; Reference address storage
D952 CHANNEL  ; Reading head address set
D954 CHANNEL  ; The start address is temporarily memorized
D956 CHANNEL  ; The data storage head address is memorized
D958 CHANNEL  ; Reading byte number set
D960 CHANNEL  ; ID4 WORKPIECE NUMBER
D966 CHANNEL  ; Number of packing in a containrt(BCD)
D967 CHANNEL  ; WORKPIECE NUMBER (BCD)
D974 CHANNEL  ; The start address is temporarily memorized
D976 CHANNEL  ; The data storage head address is memorized
D978 CHANNEL  ; Writing number of words
D980 CHANNEL  ; Writing workpiece number data
D981 CHANNEL  ; Writing equipment number data
D982 CHANNEL  ; The moon on writing clock data day
D983 CHANNEL  ; Amount at writing clock data
D986 CHANNEL  ; Number of packing in a containrt(BCD)
D987 CHANNEL  ; One lane flow workpiece number
D990 CHANNEL  ; Number of packing in a containrt(BIN)
D992 CHANNEL  ; Control data
D994 CHANNEL  ; Forwarding data
E0_110 CHANNEL  ; FAULT STOP NUMBER (WINDING No.1)
E0_111 CHANNEL  ; FLOW PRODUCT NUMBER (WINDING No.1)
E0_112 CHANNEL  ; FAULT STOP NUMBER. (WINDING No.2)
E0_113 CHANNEL  ; FLOW PRODUCT NUMBER (WINDING No.2)
E0_119 CHANNEL  ; FAULT STOP NUMBER (FUSING)
E0_120 CHANNEL  ; FIT POS DEFECT
E0_122 CHANNEL  ; CORE SLOT NG
E0_124 CHANNEL  ; CORE SLOT UPPER NG
E0_126 CHANNEL  ; CORE SLOT LOWER NG
E0_128 CHANNEL  ; PRESS FIT LOAD NG
E0_130 CHANNEL  ; PRESS FIT DIM NG
E0_132 CHANNEL  ; COMMUTATOR NG
E0_139 CHANNEL  ; FAULT STOP NUMBER (IMBALANCE CORRECTING)
E0_159 CHANNEL  ; FAULT STOP NUMBER (COMM TURNING)
E0_179 CHANNEL  ; FAULT STOP NUMBER (BURNISHING)
E0_19 CHANNEL  ; FAULT STOP NUMBER (SHAFT PRESS-FITTING)
E0_199 CHANNEL  ; FAULT STOP NUMBER (BALL STACKING)
E0_20000 CHANNEL  ; SHORT STOP DATA 1
E0_20010 CHANNEL  ; SHORT STOP DATA 2
E0_219 CHANNEL  ; FAULT STOP NUMBER (ARMATURE TESTER)
E0_23000 CHANNEL  ; SHORT STOP DATA DISPLAY
E0_23100 CHANNEL  ; Index register
E0_23102 CHANNEL  ; MEMORY NUMBER -1
E0_23104 CHANNEL  ; Data register setting
E0_23106 CHANNEL  ; Calculation register
E0_23107 CHANNEL  ; MEMORY NUMBER
E0_23200 CHANNEL  ; Operating time count
E0_23202 CHANNEL  ; Operating time (Minute and Second)
E0_23203 CHANNEL  ; Operating time (Hour)
E0_23300 CHANNEL  ; FAULT STOP MACHINE NUMBER (BIN)
E0_23301 CHANNEL  ; FAULT DISPLAY NUMBER
E0_23302 CHANNEL  ; Generation date (Month)
E0_23303 CHANNEL  ; Generation date (Day)
E0_23304 CHANNEL  ; Generation date (Hour)
E0_23305 CHANNEL  ; Generation date (Minute)
E0_23306 CHANNEL  ; SHORT STOP TIME (Hour)
E0_23307 CHANNEL  ; SHORT STOP TIME (Minute)
E0_23308 CHANNEL  ; FAULT STOP MACHINE NUMBER (BCD)
E0_23309 CHANNEL  ; PERIODICAL STOP
E0_23400 CHANNEL  ; Number of writing data
E0_23402 CHANNEL  ; Writing starting address
E0_23404 CHANNEL  ; -
E0_23405 CHANNEL  ; -
E0_23406 CHANNEL  ; Directory name & file name
E0_23407 CHANNEL  ; Directory name & file name
E0_23408 CHANNEL  ; Directory name & file name
E0_23409 CHANNEL  ; Directory name & file name
E0_250 CHANNEL  ; PROCESSING STOP
E0_25000 CHANNEL  ; STOP DATA 1
E0_25010 CHANNEL  ; STOP DATA 2
E0_252 CHANNEL  ; MEAS ROT SPD NG
E0_254 CHANNEL  ; MEAS DATA FAULT
E0_256 CHANNEL  ; INSP UNBALANCE NG
E0_258 CHANNEL  ; INSP1 ROT SPD NG
E0_260 CHANNEL  ; INSP1 DATA FAULT
E0_262 CHANNEL  ; INSP1 DATA FAULT
E0_2800 CHANNEL  ; Product number registration No. (resistance measurement ST)
E0_2813 CHANNEL  ; Master code (resistor)
E0_28300 CHANNEL  ; FAULT STOP MACHINE NUMBER (BIN)
E0_28301 CHANNEL  ; FAULT DISPLAY NUMBER
E0_28302 CHANNEL  ; Generation date (Month)
E0_28303 CHANNEL  ; Generation date (Day)
E0_28304 CHANNEL  ; Generation date (Hour)
E0_28305 CHANNEL  ; Generation date (Minute)
E0_28309 CHANNEL  ; PERIODICAL STOP
E0_28400 CHANNEL  ; Number of writing data
E0_28402 CHANNEL  ; Writing starting address
E0_28404 CHANNEL  ; -
E0_28405 CHANNEL  ; -
E0_28406 CHANNEL  ; Directory name & file name
E0_28407 CHANNEL  ; Directory name & file name
E0_28408 CHANNEL  ; Directory name & file name
E0_28409 CHANNEL  ; Directory name & file name
E0_290 CHANNEL  ; PROCESSING STOP
E0_2900 CHANNEL  ; Resistance counter electrode data 1 (180 °) (resistance)
E0_292 CHANNEL  ; MEAS ROT SPD NG
E0_294 CHANNEL  ; MEAS DATA FAULT
E0_296 CHANNEL  ; INSP UNBALANCE NG
E0_2975 CHANNEL  ; Resistance standard counter electrode lower limit (resistance)
E0_2976 CHANNEL  ; Resistance standard counter electrode upper limit (resistance)
E0_2977 CHANNEL  ; Resistance standard 180 ° Lower limit of counter electrode (resistance)
E0_2978 CHANNEL  ; Resistance standard 180 ° counter electrode upper limit (resistance)
E0_298 CHANNEL  ; INSP1 ROT SPD NG
E0_300 CHANNEL  ; INSP1 DATA FAULT
E0_30500 CHANNEL  ; Setting: Body No.
E0_310 CHANNEL  ; INSP1 DATA FAULT
E0_3200 CHANNEL  ; Part number registration No. (work reversal)
E0_3207 CHANNEL  ; With or without work (work inversion)
E0_3213 CHANNEL  ; Master data (reversing part)
E0_3400 CHANNEL  ; Product number registration No. (bearing press-fitting)
E0_3407 CHANNEL  ; Presence / absence of work (bearing press-fitting)
E0_3413 CHANNEL  ; Master data (press-fitting part)
E0_360 CHANNEL  ; Work information from the previous process (set top ADDR)
E0_3600 CHANNEL  ; Product number registration No. (total length measurement)
E0_3607 CHANNEL  ; Presence / absence of work (total length measurement)
E0_3613 CHANNEL  ; Master data (dimension measurement unit)
E0_366 CHANNEL  ; Flowing body shape information from the ball
E0_380 CHANNEL  ; CAULKING CHECK NG
E0_382 CHANNEL  ; GREASE COATING NG
E0_39 CHANNEL  ; FAULT STOP NUMBER (POWDER COATING)
E0_40 CHANNEL  ; DEFECT
E0_419 CHANNEL  ; FAULT STOP NUMBER (ARMATURE TESTER)
E0_420 CHANNEL  ; Flowing physique information
E0_425 CHANNEL  ; Currently in production Part number memory
E0_59 CHANNEL  ; FAULT STOP NUMBER (COMM PRESS-FITTING)
E0_9022 CHANNEL  ; Calculation register
E0_9024 CHANNEL  ; Calculation register
E0_9026 CHANNEL  ; Indirectly designated register
E10000 CHANNEL  ; OK DATA 1 WORKPIECE EXISTENCE
E10200 CHANNEL  ; OK DATA 2 WORKPIECE EXISTENCE
E14000 CHANNEL  ; OK DATA 1 DISPLAY WORKPIECE EXISTENCE
E15000 CHANNEL  ; NG DATA 1 WORKPIECE EXISTENCE
E15100 CHANNEL  ; -
E15200 CHANNEL  ; NG DATA 2 WORKPIECE EXISTENCE
E18999 CHANNEL  ; NG DATA 20 PRELIMINARY DATA
E19000 CHANNEL  ; NG DATA 1 DISPLAY WORKPIECE EXISTENCE
E2000 CHANNEL  ; With or Without Work
E2001 CHANNEL  ; Code No.
E2019 CHANNEL  ; Synthesis OK
E2023 CHANNEL  ; Master Check Data
E2034 CHANNEL  ; OVERALL LENGTH LOWER STANDARD VALUE
E2036 CHANNEL  ; OVERALL LENGTH UPPER STANDARD VALUE
E2040 CHANNEL  ; BEARING INSERT LENGTH LOWER STANDARD VALUE
E2042 CHANNEL  ; BEARING INSERT LENGTH UPPER STANDARD VALUE
E2058 CHANNEL  ; THICKNESS OF CORE JUDGMENT RESULT (1:L , 2: S)
E2092 CHANNEL  ; PAIR POLE RESISTANCE SPECIFICATION MINIMUM VALUE
E2093 CHANNEL  ; PAIR POLE RESISTANCE SPECIFICATION MAXIMUM VALUE
E2094 CHANNEL  ; PAIR NEXTRESISTANCE SPECIFICATION MINIMUM VALUE
E2095 CHANNEL  ; PAIR NEXT RESISTANCE SPECIFICATION MAXIMUM VALUE
E2169 CHANNEL  ; IMPULSE PAIR POLE PROGRAM No.
E2200 CHANNEL  ; WORKPIECE MEMORY
E2208 CHANNEL  ; INSULATION TEST JUDGMENT RESULT (1:OK,2:NG)
E2219 CHANNEL  ; ﾜｰｸ総合OK
E2400 CHANNEL  ; WORKPIECE MEMORY
E2408 CHANNEL  ; INSULATION TEST JUDGMENT RESULT (1:OK,2:NG)
E2415 CHANNEL  ; SWING MEASUREMENT JUDGMENT RESULT (1:OK,2:NG)
E2419 CHANNEL  ; Synthesis OK
E2448 CHANNEL  ; SHAFT END SWING JUDGMENT RESULT (1:OK,2:NG)
E2449 CHANNEL  ; WORM SWING JUDGMENT RESULT (1:OK,2:NG)
E2450 CHANNEL  ; SWINGING MEASUREMENT RESULT (SHAFT END)
E2452 CHANNEL  ; SWINGING MEASUREMENT RESULT (WORM)
E2458 CHANNEL  ; THICKNESS OF CORE JUDGMENT RESULT (1:L , 2: S)
E2459 CHANNEL  ; COIL END JUDGMENT RESULT (1:L , 2: S)
E2600 CHANNEL  ; WORKPIECE MEMORY
E2607 CHANNEL  ; UNLOADING LANE No.
E2608 CHANNEL  ; INSULATION TEST JUDGMENT RESULT (1:OK,2:NG)
E2609 CHANNEL  ; RESISTANCE MEASUREMENT JUDGMENT RESULT  (1:OK,2:NG)
E2611 CHANNEL  ; Workpiece number selection result (1:OK,2:NG)
E2614 CHANNEL  ; Temperature data (resistor)
E2615 CHANNEL  ; SWING MEASUREMENT JUDGMENT RESULT (1:OK,2:NG)
E2619 CHANNEL  ; Synthesis OK
E2620 CHANNEL  ; 80 PAIR NEXT RESISTANCE MEASUREMENT JUDGMENT RESULT (1:OK,2:NG)
E2621 CHANNEL  ; 180 PAIR  RESISTANCE MEASUREMENT JUDGMENT RESULT (1:OK,2:NG)
E2634 CHANNEL  ; OVERALL LENGTH LOWER STANDARD VALUE
E2640 CHANNEL  ; BEARING INSERT LENGTH LOWER STANDARD VALUE
E2658 CHANNEL  ; THICKNESS OF CORE JUDGMENT RESULT (1:L , 2: S)
E2659 CHANNEL  ; COIL END JUDGMENT RESULT (1:L , 2: S)
E2664 CHANNEL  ; NUMBER OF TURNS RESULT (1:L , 2:H , 3:NG)
E2670 CHANNEL  ; PAIR POLE RESISTANCE MEASUREMENT DATA 1
E2692 CHANNEL  ; PAIR POLE RESISTANCE SPECIFICATION MINIMUM VALUE
E2693 CHANNEL  ; PAIR POLE RESISTANCE SPECIFICATION MAXIMUM VALUE
E2766 CHANNEL  ; IMPULSE NEXT POLE PAGE No.
E2800 CHANNEL  ; WORKPIECE MEMORY
E2808 CHANNEL  ; INSULATION TEST JUDGMENT RESULT (1:OK,2:NG)
E2809 CHANNEL  ; RESISTANCE MEASUREMENT JUDGMENT RESULT (1:OK,2:NG)
E2810 CHANNEL  ; IMPULSE MEASUREMENT JUDGMENT RESULT (1:OK,2:NG)
E2811 CHANNEL  ; Workpiece number selection result (1:OK,2:NG)
E2812 CHANNEL  ; IMPULSE NEXT POLE JUDGMENT RESULT (1:OK,2:NG)
E2813 CHANNEL  ; IMPULSE PAIR POLE JUDGMENT RESULT (1:OK,2:NG)
E2815 CHANNEL  ; SWING MEASUREMENT JUDGMENT RESULT (1:OK,2:NG)
E2819 CHANNEL  ; Synthesis OK
E2823 CHANNEL  ; Master data (impulse section)
E2966 CHANNEL  ; IMPULSE NEXT POLE PAGE No.
E2967 CHANNEL  ; IMPULSE NEXT POLE PROGRAM No.
E2968 CHANNEL  ; IMPULSE PAIR POLE PAGE No.
E2969 CHANNEL  ; IMPULSE PAIR POLE PROGRAM No.
E3000 CHANNEL  ; WORKPIECE MEMORY
E3008 CHANNEL  ; INSULATION TEST JUDGMENT RESULT (1:OK,2:NG)
E3009 CHANNEL  ; RESISTANCE MEASUREMENT JUDGMENT RESULT (1:OK,2:NG)
E3010 CHANNEL  ; IMPULSE MEASUREMENT JUDGMENT RESULT (1:OK,2:NG)
E3011 CHANNEL  ; Workpiece number selection result (1:OK,2:NG)
E3015 CHANNEL  ; SWING MEASUREMENT JUDGMENT RESULT (1:OK,2:NG)
E3019 CHANNEL  ; Synthesis OK
E3046 CHANNEL  ; PRESENCE OF INSERT (1: No , 2: Having)
E3060 CHANNEL  ; BEARING INSERT JUDGMENT RESULT (1:OK,2:NG)
E3200 CHANNEL  ; WORKPIECE MEMORY
E3208 CHANNEL  ; INSULATION TEST JUDGMENT RESULT (1:OK,2:NG)
E3209 CHANNEL  ; RESISTANCE MEASUREMENT JUDGMENT RESULT (1:OK,2:NG)
E3210 CHANNEL  ; IMPULSE MEASUREMENT JUDGMENT RESULT (1:OK,2:NG)
E3211 CHANNEL  ; Workpiece number selection result (1:OK,2:NG)
E3215 CHANNEL  ; SWING MEASUREMENT JUDGMENT RESULT (1:OK,2:NG)
E3216 CHANNEL  ; LENGTH MEASUREMENT JUDGMENT RESULT (1:OK,2:NG)
E3219 CHANNEL  ; Synthesis OK
E3223 CHANNEL  ; Master data
E3234 CHANNEL  ; OVERALL LENGTH LOWER STANDARD VALUE
E3236 CHANNEL  ; OVERALL LENGTH UPPER STANDARD VALUE
E3240 CHANNEL  ; BEARING INSERT LENGTH LOWER STANDARD VALUE
E3242 CHANNEL  ; BEARING INSERT LENGTH UPPER STANDARD VALUE
E3246 CHANNEL  ; PRESENCE OF INSERT (1: No , 2: Having)
E3254 CHANNEL  ; LENGTH MEASUREMENT DATA (OVERALL)
E3256 CHANNEL  ; LENGTH MEASUREMENT DATA (BEARING)
E3260 CHANNEL  ; BEARING INSERT JUDGMENT RESULT (1:OK,2:NG)
E3261 CHANNEL  ; LENGTH MEASUREMENT JUDGMENT RESULT (1:OK,2:NG)
E3262 CHANNEL  ; BEARING INSERT MEASUREMENT  JUDGMENT RESULT (1:OK,2:NG)
E3400 CHANNEL  ; WORKPIECE MEMORY
E3419 CHANNEL  ; Synthesis OK
E3569 CHANNEL  ; IMPULSE PAIR POLE PROGRAM No.
E3600 CHANNEL  ; WORKPIECE MEMORY
E3601 CHANNEL  ; CODE No.
E3608 CHANNEL  ; INSULATION TEST JUDGMENT RESULT (1:OK,2:NG)
E3609 CHANNEL  ; RESISTANCE MEASUREMENT JUDGMENT RESULT (1:OK,2:NG)
E3610 CHANNEL  ; IMPULSE MEASUREMENT JUDGMENT RESULT (1:OK,2:NG)
E3611 CHANNEL  ; Workpiece number selection result (1:OK,2:NG)
E3615 CHANNEL  ; SWING MEASUREMENT JUDGMENT RESULT (1:OK,2:NG)
E3616 CHANNEL  ; LENGTH MEASUREMENT JUDGMENT RESULT (1:OK,2:NG)
E3619 CHANNEL  ; Synthesis OK
E3661 CHANNEL  ; LENGTH MEASUREMENT JUDGMENT RESULT (1:OK,2:NG)
E3662 CHANNEL  ; BEARING INSERT MEASUREMENT  JUDGMENT RESULT (1:OK,2:NG)
E3769 CHANNEL  ; IMPULSE PAIR POLE PROGRAM No.
E3800 CHANNEL  ; WORKPIECE MEMORY
E4000 CHANNEL  ; WORKPIECE MEMORY
E4169 CHANNEL  ; IMPULSE PAIR POLE PROGRAM No.
E5400 CHANNEL  ; WORKPIECE MEMORY
E5569 CHANNEL  ; IMPULSE PAIR POLE PROGRAM No.
E6005 CHANNEL  ; PAIR POLE RESISTANCE MEASUREMENT DATA 1
E6035 CHANNEL  ; PAIR POLE RESISTANCE MEASUREMENT DATA 1
E6036 CHANNEL  ; PAIR POLE RESISTANCE MEASUREMENT DATA 1
E6065 CHANNEL  ; PAIR POLE RESISTANCE SPECIFICATION MINIMUM VALUE
E6066 CHANNEL  ; PAIR POLE RESISTANCE SPECIFICATION MAXIMUM VALUE
E6095 CHANNEL  ; PAIR POLE RESISTANCE SPECIFICATION MINIMUM VALUE
E6096 CHANNEL  ; PAIR POLE RESISTANCE SPECIFICATION MAXIMUM VALUE
E6125 CHANNEL  ; PAIR POLE RESISTANCE SPECIFICATION MINIMUM VALUE
E6126 CHANNEL  ; PAIR POLE RESISTANCE SPECIFICATION MAXIMUM VALUE
E6155 CHANNEL  ; PAIR POLE RESISTANCE SPECIFICATION MINIMUM VALUE
E6156 CHANNEL  ; PAIR POLE RESISTANCE SPECIFICATION MAXIMUM VALUE
E6185 CHANNEL  ; PAIR POLE RESISTANCE SPECIFICATION MINIMUM VALUE
E6186 CHANNEL  ; PAIR POLE RESISTANCE SPECIFICATION MAXIMUM VALUE
E6215 CHANNEL  ; PAIR POLE RESISTANCE MEASUREMENT DATA 1
E6216 CHANNEL  ; PAIR POLE RESISTANCE MEASUREMENT DATA 1
E6245 CHANNEL  ; PAIR POLE RESISTANCE MEASUREMENT DATA 1
E6246 CHANNEL  ; PAIR POLE RESISTANCE MEASUREMENT DATA 1
E6900 CHANNEL  ; LANE 1 WORKPIECE NUMBER
E6901 CHANNEL  ; LANE 2 WORKPIECE NUMBER
E6902 CHANNEL  ; LANE 1 WORKPIECE PRODUCT NUMBER
E6903 CHANNEL  ; LANE 2 WORKPIECE PRODUCT NUMBER
E7000 CHANNEL  ; CODE No. (LANE 1)
E7030 CHANNEL  ; CODE No. (LANE 2)
E8000 CHANNEL  ; Calculation register
E8002 CHANNEL  ; -
E8004 CHANNEL  ; Register of indirect specification
E8006 CHANNEL  ; -
E8020 CHANNEL  ; CODE No.
E8022 CHANNEL  ; Calculation register
E8024 CHANNEL  ; Calculation register
E8026 CHANNEL  ; Register of indirect specification
E9100 CHANNEL  ; OK DATA INDEX REGISTER
E9102 CHANNEL  ; CALCULATION REGISTER
E9104 CHANNEL  ; DATA REGISTER SET UP
E9106 CHANNEL  ; CALCULATION REGISTER
E9107 CHANNEL  ; -
E9120 CHANNEL  ; DEFECTIVE INDEX REGISTER
E9122 CHANNEL  ; CALCULATION REGISTER
E9124 CHANNEL  ; DATA REGISTER SET UP
E9126 CHANNEL  ; CALCULATION REGISTER
E9127 CHANNEL  ; CALCULATION REGISTER
E9263 CHANNEL  ; SPECIFICATION VALUE ADDRESS INDIRECT SPECIFICATION
E9280 CHANNEL  ; SPECIFICATION VALUE ADDRESS INDIRECT SPECIFICATION
E9304 CHANNEL  ; Standard value comparison result 1
E9306 CHANNEL  ; Standard value comparison result 2 (After the mask)
H0.02 BOOL  ; XXXX
H0.04 BOOL  ; NG WORKPIECE INSULATION TEST
H0.05 BOOL  ; NG WORKPIECE IMPULSE MEASURE
H0.06 BOOL  ; NG WORKPIECE SWING MEASURE
H0.07 BOOL  ; NG WORKPIECE BEARING INSERT
H0.08 BOOL  ; NG WORKPIECE RESISTANCE MEASURE
H0.09 BOOL  ; NG WORKPIECE LENGTH MEASURE
H0.10 BOOL  ; LANE 1 CONFIRMATION THE OPERATION
H0.11 BOOL  ; LANE 2 CONFIRMATION THE OPERATION
H0.12 BOOL  ; ID INVALIDITY OPERATION
H10.00 BOOL  ; ID RESET START SELECT OF LANE 1
H110 CHANNEL  ; 01ST_STEP
H110.00 BOOL  ; 01ST_STEP START
H110.01 BOOL  ; 01ST_STEP 01
H110.02 BOOL  ; 01ST_STEP 02
H110.03 BOOL  ; 01ST_STEP 03
H110.04 BOOL  ; 01ST_STEP 04
H115 CHANNEL  ; 02ST_STEP
H115.00 BOOL  ; 02ST_STEP START
H115.01 BOOL  ; 02ST_STEP 02
H115.02 BOOL  ; 02ST_STEP 02
H115.03 BOOL  ; 02ST_STEP 03
H115.04 BOOL  ; 02ST_STEP 04
H115.05 BOOL  ; 02ST_STEP 05
H115.06 BOOL  ; 02ST_STEP 06
H115.07 BOOL  ; 02ST_STEP 07
H115.08 BOOL  ; 02ST_STEP 08
H115.09 BOOL  ; 02ST_STEP 09
H115.10 BOOL  ; 02ST_STEP 10
H120 CHANNEL  ; 03ST_STEP
H120.00 BOOL  ; 03ST_STEP START_1 Cycle Preparation
H120.01 BOOL  ; 03ST_STEP 03_Transfer Unit FWD
H120.02 BOOL  ; 03ST_STEP 02_WorkPiece Clamp Down Good Condition for other process
H120.03 BOOL  ; 03ST_STEP 03_Workpiece Clamp Signal Transfer Complet
H120.04 BOOL  ; 03ST_STEP 04_Waiting WorkPiece Clam Down Complete
H120.05 BOOL  ; 03ST_STEP 05_Transfer Carrier Up
H120.06 BOOL  ; 03ST_STEP 06_Measuring Good Condition Signal for other process
H120.07 BOOL  ; 03ST_STEP 07_Measuring Good Condition Signal for other process Transfer Complete
H120.08 BOOL  ; 03ST_STEP 08_Transfer Carrier BWD Waiting Good Condition
H120.09 BOOL  ; 03ST_STEP 09
H120.10 BOOL  ; 03ST_STEP 10
H120.11 BOOL  ; 03ST_STEP 11
H120.12 BOOL  ; 03ST_STEP 12
H120.13 BOOL  ; 03ST_STEP 13
H120.14 BOOL  ; 03ST_STEP 14
H125 CHANNEL  ; 04ST_STEP
H125.00 BOOL  ; 04ST_STEP START
H125.01 BOOL  ; 04ST_STEP 04
H125.02 BOOL  ; 04ST_STEP 02
H125.03 BOOL  ; 04ST_STEP 03
H125.04 BOOL  ; 04ST_STEP 04
H130 CHANNEL  ; 05ST_STEP
H130.00 BOOL  ; 05ST_STEP START
H130.01 BOOL  ; 05ST_STEP 05
H130.02 BOOL  ; 05ST_STEP 02
H130.03 BOOL  ; 05ST_STEP 03
H130.04 BOOL  ; 05ST_STEP 04
H130.05 BOOL  ; 05ST_STEP 05
H130.06 BOOL  ; 05ST_STEP 06
H130.07 BOOL  ; 05ST_STEP 07
H130.14 BOOL  ; 05ST_STEP 14
H130.15 BOOL  ; 05ST_STEP 15
H131 CHANNEL  ; 05ST_STEP
H135 CHANNEL  ; 06ST_STEP
H135.00 BOOL  ; 06ST_STEP START
H135.01 BOOL  ; 06ST_STEP 06
H135.02 BOOL  ; 06ST_STEP 02
H135.03 BOOL  ; 06ST_STEP 03
H135.04 BOOL  ; 06ST_STEP 04
H135.05 BOOL  ; 06ST_STEP 05
H135.06 BOOL  ; 06ST_STEP 06
H135.07 BOOL  ; 06ST_STEP 07
H135.08 BOOL  ; 06ST_STEP 08
H135.09 BOOL  ; 06ST_STEP 09
H135.10 BOOL  ; 06ST_STEP 10
H135.11 BOOL  ; 06ST_STEP 11
H135.12 BOOL  ; 06ST_STEP 12
H135.13 BOOL  ; 06ST_STEP 13
H135.14 BOOL  ; 06ST_STEP 14
H135.15 BOOL  ; 06ST_STEP 15
H140 CHANNEL  ; 07ST_STEP
H140.00 BOOL  ; 07ST_STEP START
H140.01 BOOL  ; 07ST_STEP 07_Work Piece Down Clamp Signal Good Condition Check
H140.02 BOOL  ; 07ST_STEP 02_Work Piece Down Clamp Signal Good Condition Check Confirm
H140.03 BOOL  ; 07ST_STEP 03_Workpiece Ready Check
H140.04 BOOL  ; 07ST_STEP 04_WorkPiece Clam Down
H140.05 BOOL  ; 07ST_STEP 05_Measuring Good Condition Signal Waiting
H140.06 BOOL  ; 07ST_STEP 06_Measuring Good Condition Signal Complete
H140.07 BOOL  ; 07ST_STEP 07
H140.08 BOOL  ; 07ST_STEP 08
H140.09 BOOL  ; 07ST_STEP 09_Workpiece Check Before Measuring
H140.10 BOOL  ; 07ST_STEP 10_Contact Probe FWD
H140.11 BOOL  ; 07ST_STEP 11
H140.12 BOOL  ; 07ST_STEP 12
H140.13 BOOL  ; 07ST_STEP 13_Probe BWD
H140.14 BOOL  ; 07ST_STEP 14
H140.15 BOOL  ; 07ST_STEP 15
H145 CHANNEL  ; ST8_Impulse measurement unit_step circuit
H145.00 BOOL  ; 08ST_STEP START_1 Cycle Preparation
H145.01 BOOL  ; 08ST_STEP 08_Work Piece Down Clamp Signal Good Condition Check
H145.02 BOOL  ; 08ST_STEP 02_Work Piece Down Clamp Signal Good Condition Check Confirm
H145.03 BOOL  ; 08ST_STEP 03_Workpiece Ready Check
H145.04 BOOL  ; 08ST_STEP 04_WorkPiece Clam Down
H145.05 BOOL  ; 08ST_STEP 05_Measuring Good Condition Signal Waiting
H145.06 BOOL  ; 08ST_STEP 06_Measuring Good Condition Signal Complete
H145.07 BOOL  ; 08ST_STEP 07
H145.08 BOOL  ; 08ST_STEP 08
H145.09 BOOL  ; 08ST_STEP 09_Workpiece Check
H145.10 BOOL  ; 08ST_STEP 10_Contact Probe FWD
H145.11 BOOL  ; 08ST_STEP 11_Impulse Check
H145.12 BOOL  ; 08ST_STEP 12_Probe BWD (Measuring Complete)
H145.13 BOOL  ; 08ST_STEP 13
H145.14 BOOL  ; 08ST_STEP 14
H145.15 BOOL  ; 08ST_STEP 15
H146 CHANNEL  ; IMPULSE_STEP
H146.00 BOOL  ; IMPULSE_STEP START
H146.01 BOOL  ; IMPULSE_STEP 01
H146.02 BOOL  ; IMPULSE_STEP 02
H146.03 BOOL  ; IMPULSE_STEP 03
H146.04 BOOL  ; IMPULSE_STEP 04
H146.05 BOOL  ; IMPULSE_STEP 05
H146.06 BOOL  ; IMPULSE_STEP 06
H146.07 BOOL  ; IMPULSE_STEP 07
H146.08 BOOL  ; IMPULSE_STEP 08
H146.09 BOOL  ; IMPULSE_STEP 09
H146.10 BOOL  ; IMPULSE_STEP 10
H146.11 BOOL  ; IMPULSE_STEP 11
H146.12 BOOL  ; IMPULSE_STEP 12
H146.13 BOOL  ; IMPULSE_STEP 13
H146.14 BOOL  ; IMPULSE_STEP 14
H146.15 BOOL  ; IMPULSE_STEP 15
H147 CHANNEL  ; Impulse analysis step circuit
H147.00 BOOL  ; Impals_Analysis Step 00
H147.01 BOOL  ; Impals_Analysis Step 01
H147.02 BOOL  ; Impulse_Analysis Step 02
H147.03 BOOL  ; Impulse_Analysis Step 03
H147.04 BOOL  ; Impulse_Analysis Step 04
H147.05 BOOL  ; Impulse_Analysis Step 05
H147.06 BOOL  ; Impulse_Analysis Step 06
H147.07 BOOL  ; Impulse_Analysis Step 07
H150 CHANNEL  ; 09ST_STEP
H150.00 BOOL  ; 09ST_STEP START
H150.01 BOOL  ; 09ST_STEP 09
H150.02 BOOL  ; 09ST_STEP 02
H150.03 BOOL  ; 09ST_STEP 03
H150.04 BOOL  ; 09ST_STEP 04
H150.05 BOOL  ; 09ST_STEP 05
H150.06 BOOL  ; 09ST_STEP 06
H150.07 BOOL  ; 09ST_STEP 07
H150.08 BOOL  ; 09ST_STEP 08
H150.09 BOOL  ; 09ST_STEP 09
H150.10 BOOL  ; 09ST_STEP 10
H150.11 BOOL  ; 09ST_STEP 11
H150.12 BOOL  ; 09ST_STEP 12
H150.15 BOOL  ; 09ST_STEP 15
H151.00 BOOL  ; step0 Bearing press-fit work press down
H151.01 BOOL  ; step1 Guide advance
H151.02 BOOL  ; step2 Bearing press-fit work presser rise
H151.03 BOOL  ; step3 Press-fit forward
H151.04 BOOL  ; step4 Press-fit retreat
H151.05 BOOL  ; step5 Bearing press-fit work press down
H151.06 BOOL  ; step6 Bearing guide receding end
H151.07 BOOL  ; Bearing press-fit work presser rise
H155 CHANNEL  ; 10ST_STEP
H155.00 BOOL  ; 10ST_STEP START
H155.01 BOOL  ; 10ST_STEP 10
H155.02 BOOL  ; 10ST_STEP 02
H155.03 BOOL  ; 10ST_STEP 03
H155.04 BOOL  ; 10ST_STEP 04
H155.05 BOOL  ; 10ST_STEP 05
H155.06 BOOL  ; 10ST_STEP 06
H155.07 BOOL  ; 10ST_STEP 07
H155.08 BOOL  ; 10ST_STEP 08
H155.09 BOOL  ; -
H155.15 BOOL  ; 10ST_STEP 15
H157 CHANNEL  ; MASTER SET_STEP
H157.00 BOOL  ; MASTER SET_STEP START
H157.01 BOOL  ; MASTER SET_STEP 01
H157.02 BOOL  ; MASTER SET_STEP 02
H157.03 BOOL  ; MASTER SET_STEP 03
H157.04 BOOL  ; MASTER SET_STEP 04
H157.05 BOOL  ; MASTER SET_STEP 05
H157.06 BOOL  ; MASTER SET_STEP 06
H157.07 BOOL  ; MASTER SET_STEP 07
H157.08 BOOL  ; MASTER SET_STEP 08
H159 CHANNEL  ; Upper limit Master check circuit
H159.00 BOOL  ; Master 0
H159.01 BOOL  ; Master 1
H159.02 BOOL  ; Master 2
H159.03 BOOL  ; Master 3
H159.04 BOOL  ; Master 6 measuring element forward
H159.05 BOOL  ; Upper limit check steffe 5 (functional check)
H159.06 BOOL  ; Master 6 measuring element retreat
H159.07 BOOL  ; Master 7 Measurement position confirmation Upper limit inspection
H159.08 BOOL  ; Master 8 measuring element retreat
H160 CHANNEL  ; 11ST_STEP
H160.00 BOOL  ; 11ST_STEP START
H160.01 BOOL  ; 11ST_STEP 11
H160.02 BOOL  ; 11ST_STEP 02
H160.03 BOOL  ; 11ST_STEP 03
H160.04 BOOL  ; 11ST_STEP 04
H160.05 BOOL  ; 11ST_STEP 05
H160.06 BOOL  ; 11ST_STEP 06
H160.07 BOOL  ; 11ST_STEP 07
H160.08 BOOL  ; 11ST_STEP 08
H160.09 BOOL  ; 11ST_STEP 09
H160.10 BOOL  ; 11ST_STEP 10
H160.11 BOOL  ; 11ST_STEP 11
H160.15 BOOL  ; 11ST_STEP 15
H162 CHANNEL  ; Lower limit check step circuit (functional check)
H162.00 BOOL  ; Lower limit check step circuit (functional check)
H162.01 BOOL  ; Lower limit check step circuit (functional check)
H162.02 BOOL  ; Lower limit check step circuit (functional check)
H162.03 BOOL  ; Lower limit check step circuit (functional check)
H162.04 BOOL  ; Lower limit check step circuit (functional check)
H162.05 BOOL  ; Lower limit check step circuit (functional check)
H162.06 BOOL  ; Lower limit check step circuit (functional check)
H162.07 BOOL  ; Lower limit check step circuit (functional check)
H162.08 BOOL  ; Lower limit check step circuit (functional check)
H165 CHANNEL  ; 12ST_STEP
H165.00 BOOL  ; 12ST_STEP START
H165.01 BOOL  ; 12ST_STEP 12
H165.02 BOOL  ; 12ST_STEP 02
H165.03 BOOL  ; 12ST_STEP 03
H165.04 BOOL  ; 12ST_STEP 04
H165.05 BOOL  ; 12ST_STEP 05
H165.06 BOOL  ; 12ST_STEP 06
H165.07 BOOL  ; 12ST_STEP 07
H165.08 BOOL  ; 12ST_STEP 08
H165.09 BOOL  ; 12ST_STEP 09
H165.10 BOOL  ; 12ST_STEP 10
H165.11 BOOL  ; 12ST_STEP 11
H165.12 BOOL  ; 12ST_STEP 12
H165.13 BOOL  ; 12ST_STEP 13
H165.14 BOOL  ; 12ST_STEP 14
H165.15 BOOL  ; 12ST_STEP 15
H166.00 BOOL  ; 12ST_STEP 16
H166.01 BOOL  ; 12ST_STEP 17
H166.02 BOOL  ; 12ST_STEP 18
H170 CHANNEL  ; 13ST_STEP
H170.00 BOOL  ; 13ST_STEP START
H170.01 BOOL  ; 13ST_STEP 13
H170.02 BOOL  ; 13ST_STEP 02
H170.03 BOOL  ; 13ST_STEP 03
H170.04 BOOL  ; 13ST_STEP 04
H170.05 BOOL  ; 13ST_STEP 05
H170.06 BOOL  ; 13ST_STEP 06
H170.07 BOOL  ; 13ST_STEP 07
H170.08 BOOL  ; 13ST_STEP 08
H170.09 BOOL  ; 13ST_STEP 09
H170.10 BOOL  ; 13ST_STEP 10
H170.11 BOOL  ; 13ST_STEP 11
H170.12 BOOL  ; 13ST_STEP 12
H170.13 BOOL  ; 13ST_STEP 13
H170.14 BOOL  ; 13ST_STEP 14
H170.15 BOOL  ; 13ST_STEP 15
H175 CHANNEL  ; 14ST_STEP
H175.00 BOOL  ; 14ST_STEP START
H175.01 BOOL  ; 14ST_STEP 14
H175.02 BOOL  ; 14ST_STEP 02
H175.03 BOOL  ; 14ST_STEP 03
H180 CHANNEL  ; 15ST_STEP
H180.00 BOOL  ; 15ST_STEP START
H180.01 BOOL  ; 15ST_STEP 15
H180.02 BOOL  ; 15ST_STEP 02
H180.03 BOOL  ; 15ST_STEP 03
H180.04 BOOL  ; 15ST_STEP 04
H180.05 BOOL  ; 15ST_STEP 05
H180.06 BOOL  ; 15ST_STEP 06
H180.07 BOOL  ; 15ST_STEP 07
H180.08 BOOL  ; 15ST_STEP 08
H180.09 BOOL  ; 15ST_STEP 09
H180.10 BOOL  ; 15ST_STEP 10
H180.11 BOOL  ; 15ST_STEP 11
H180.12 BOOL  ; 15ST_STEP 12
H180.13 BOOL  ; 15ST_STEP 13
H180.14 BOOL  ; 15ST_STEP 14
H180.15 BOOL  ; 15ST_STEP 15
H181 CHANNEL  ; 15ST_STEP
H181.00 BOOL  ; 15ST_STEP 16
H181.01 BOOL  ; 15ST_STEP 17
H181.02 BOOL  ; 15ST_STEP 18
H181.03 BOOL  ; 15ST_STEP 19
H181.04 BOOL  ; 15ST_STEP 20
H185 CHANNEL  ; 16ST_STEP
H185.00 BOOL  ; 16ST_STEP START
H185.01 BOOL  ; 16ST_STEP 16
H185.02 BOOL  ; 16ST_STEP 02
H185.03 BOOL  ; 16ST_STEP 03
H185.04 BOOL  ; 16ST_STEP 04
H185.05 BOOL  ; 16ST_STEP 05
H185.06 BOOL  ; 16ST_STEP 06
H185.07 BOOL  ; 16ST_STEP 07
H185.08 BOOL  ; 16ST_STEP 08
H185.09 BOOL  ; 16ST_STEP 09
H185.10 BOOL  ; 16ST_STEP 10
H185.11 BOOL  ; 16ST_STEP 11
H185.12 BOOL  ; 16ST_STEP 12
H190 CHANNEL  ; 17ST_STEP
H190.00 BOOL  ; 17ST_STEP START
H190.01 BOOL  ; 17ST_STEP 17
H190.02 BOOL  ; 17ST_STEP 02
H190.03 BOOL  ; 17ST_STEP 03
H190.04 BOOL  ; 17ST_STEP 04
H190.05 BOOL  ; 17ST_STEP 05
H190.06 BOOL  ; 17ST_STEP 06
H190.07 BOOL  ; 17ST_STEP 07
H190.08 BOOL  ; 17ST_STEP 08
H190.09 BOOL  ; 17ST_STEP 09
H190.10 BOOL  ; 17ST_STEP 10
H190.11 BOOL  ; 17ST_STEP 11
H190.12 BOOL  ; 17ST_STEP 12
H190.13 BOOL  ; 17ST_STEP 13
H190.14 BOOL  ; 17ST_STEP 14
H190.15 BOOL  ; 17ST_STEP 15
H191 CHANNEL  ; 17ST_STEP
H191.00 BOOL  ; 17ST_STEP 16
H191.01 BOOL  ; 17ST_STEP 17
H191.02 BOOL  ; 17ST_STEP 18
H191.03 BOOL  ; 17ST_STEP 19
H195 CHANNEL  ; 18ST_STEP
H195.00 BOOL  ; 18ST_STEP START
H195.01 BOOL  ; 18ST_STEP 18
H195.02 BOOL  ; 18ST_STEP 02
H195.03 BOOL  ; 18ST_STEP 03
H195.04 BOOL  ; 18ST_STEP 04
H195.05 BOOL  ; 18ST_STEP 05
H195.06 BOOL  ; 18ST_STEP 06
H195.07 BOOL  ; 18ST_STEP 07
H195.08 BOOL  ; 18ST_STEP 08
H195.09 BOOL  ; 18ST_STEP 09
H195.10 BOOL  ; 18ST_STEP 10
H195.11 BOOL  ; 18ST_STEP 11
H195.12 BOOL  ; 18ST_STEP 12
H195.13 BOOL  ; 18ST_STEP 13
H195.14 BOOL  ; 18ST_STEP 14
H195.15 BOOL  ; 18ST_STEP 15
H196.00 BOOL  ; 18ST_STEP 16
H196.01 BOOL  ; 18ST_STEP 17
H196.02 BOOL  ; 18ST_STEP 18
H196.03 BOOL  ; 18ST_STEP 19
H196.04 BOOL  ; 18ST_STEP 20
H200 CHANNEL  ; 19ST_STEP
H200.00 BOOL  ; 19ST_STEP START
H200.01 BOOL  ; 19ST_STEP 19
H200.02 BOOL  ; 19ST_STEP 02
H200.03 BOOL  ; 19ST_STEP 03
H200.04 BOOL  ; 19ST_STEP 04
H200.05 BOOL  ; 19ST_STEP 05
H200.06 BOOL  ; 19ST_STEP 06
H200.07 BOOL  ; 19ST_STEP 07
H200.08 BOOL  ; 19ST_STEP 08
H200.09 BOOL  ; 19ST_STEP 09
H200.10 BOOL  ; 19ST_STEP 10
H200.11 BOOL  ; 19ST_STEP 11
H200.12 BOOL  ; 19ST_STEP 12
H205 CHANNEL  ; 20ST_STEP
H205.00 BOOL  ; 20ST_STEP START
H205.01 BOOL  ; 20ST_STEP 20
H205.02 BOOL  ; 20ST_STEP 02
H205.03 BOOL  ; 20ST_STEP 03
H205.04 BOOL  ; 20ST_STEP 04
H205.05 BOOL  ; 20ST_STEP 05
H205.06 BOOL  ; 20ST_STEP 06
H205.07 BOOL  ; 20ST_STEP 07
H205.08 BOOL  ; 20ST_STEP 08
H205.09 BOOL  ; 20ST_STEP 09
H205.10 BOOL  ; 20ST_STEP 10
H205.11 BOOL  ; 20ST_STEP 11
H205.12 BOOL  ; 20ST_STEP 12
H205.13 BOOL  ; 20ST_STEP 13
H205.14 BOOL  ; 20ST_STEP 14
H205.15 BOOL  ; 20ST_STEP 15
H206 CHANNEL  ; 20ST_STEP
H206.00 BOOL  ; 20ST_STEP 16
H206.01 BOOL  ; 20ST_STEP 17
H206.02 BOOL  ; 20ST_STEP 18
H206.03 BOOL  ; 20ST_STEP 19
H21.00 BOOL  ; INITIAL SETTING AT MASTER ON
H280.00 BOOL  ; -
H280.10 BOOL  ; Confirmation of completion of LM physique switching
H280.11 BOOL  ; Confirmation of completion of S physique switching
H317.00 BOOL  ; LOADER CLAMP MEMORY
H325.00 BOOL  ; 04ST_COMPLETE
H326.00 BOOL  ; PUSHING WORKPIECE
H330.00 BOOL  ; 05ST_COMPLETE
H331.00 BOOL  ; INSULATION WORKPIECE
H331.02 BOOL  ; Synthesis OK
H331.03 BOOL  ; Synthesis NG
H331.04 BOOL  ; INSULATION OK
H331.05 BOOL  ; INSULATION NG
H331.06 BOOL  ; 7st operation disabled (valid at master)
H331.07 BOOL  ; With Insulation resistant master
H331.08 BOOL  ; OK WORKPIECE
H335.00 BOOL  ; 06ST_COMPLETE
H336.00 BOOL  ; SWING WORKPIECE
H336.02 BOOL  ; Synthesis OK
H336.03 BOOL  ; Synthesis NG
H336.04 BOOL  ; SWING MEASUREMENT OK
H336.05 BOOL  ; SWING MEASUREMENT NG
H336.06 BOOL  ; 6st operation disabled (valid at master)
H336.07 BOOL  ; 振れ部ﾏｽﾀｰﾜｰｸ有り
H336.08 BOOL  ; OK WORKPIECE
H336.09 BOOL  ; There is a tip runout master work
H336.10 BOOL  ; There is a warm shake master work
H340.00 BOOL  ; 07ST_COMPLETE
H341.00 BOOL  ; RESISTANCE WORKPIECE
H341.02 BOOL  ; Synthesis OK
H341.03 BOOL  ; Synthesis NG
H341.04 BOOL  ; 80 RESISTANCE MEASUREMENT OK
H341.05 BOOL  ; 80 RESISTANCE MEASUREMENT NG
H341.06 BOOL  ; WORK No. OK
H341.07 BOOL  ; WORK No. NG
H341.08 BOOL  ; OK WORKPIECE
H341.10 BOOL  ; $?St$Bk?_#[19] / NUMBER OF TURNS "L"$?St$Bk?_#[19]
H341.11 BOOL  ; $?St$Bk?_#[20] / NUMBER OF TURNS "H"$?St$Bk?_#[20]
H341.12 BOOL  ; $?St$Bk?_#[21] / NUMBER OF TURNS "NG"$?St$Bk?_#[21]
H341.13 BOOL  ; 3rd resistance master check
H341.14 BOOL  ; 4th resistance master check
H342 CHANNEL  ; PAIR RESISTANCE MEASUREMENT OK
H342.00 BOOL  ; PAIR RESISTANCE 1 OK
H342.01 BOOL  ; PAIR RESISTANCE 2 OK
H342.02 BOOL  ; PAIR RESISTANCE 3 OK
H342.03 BOOL  ; PAIR RESISTANCE 4 OK
H342.04 BOOL  ; PAIR RESISTANCE 5 OK
H342.05 BOOL  ; PAIR RESISTANCE 6 OK
H342.06 BOOL  ; Counter electrode resistance 7OK
H342.07 BOOL  ; Counter electrode resistance 8OK
H342.08 BOOL  ; Counter electrode resistance 9OK
H343 CHANNEL  ; PAIR RESISTANCE MEASUREMENT NG
H343.00 BOOL  ; PAIR RESISTANCE 1 NG
H343.01 BOOL  ; PAIR RESISTANCE 2 NG
H343.02 BOOL  ; PAIR RESISTANCE 3 NG
H343.03 BOOL  ; PAIR RESISTANCE 4 NG
H343.04 BOOL  ; PAIR RESISTANCE 5 NG
H343.05 BOOL  ; PAIR RESISTANCE 6 NG
H343.06 BOOL  ; Counter electrode resistance 7NG
H343.07 BOOL  ; Counter electrode resistance 8NG
H343.08 BOOL  ; Counter electrode resistance 9NG
H344.00 BOOL  ; 7st operation disabled (valid at master)
H344.01 BOOL  ; 1st resistance master check
H344.02 BOOL  ; Second resistance master check
H344.03 BOOL  ; 3rd resistance master check
H344.04 BOOL  ; 4th resistance master check
H344.10 BOOL  ; With resistance part master work
H345.00 BOOL  ; 08ST_COMPLETE
H346.00 BOOL  ; IMPULSE WORKPIECE
H346.02 BOOL  ; Synthesis OK
H346.03 BOOL  ; Synthesis NG
H346.04 BOOL  ; PAIR POLE OK
H346.05 BOOL  ; PAIR POLE NG
H346.06 BOOL  ; NEXT POLE OK
H346.07 BOOL  ; NEXT POLE NG
H346.08 BOOL  ; OKﾜｰｸ
H346.09 BOOL  ; 8st operation disabled (valid at master)
H346.10 BOOL  ; Impulse part with master work
H346.11 BOOL  ; Impulse Master 1st
H346.12 BOOL  ; Impulse Master 2nd
H346.13 BOOL  ; Impulse Master 3rd
H347.00 BOOL  ; 180 RESISTANCE MEASUREMENT OK
H347.01 BOOL  ; 180 RESISTANCE MEASUREMENT NG
H351.00 BOOL  ; INSERT WORKPIECE
H351.02 BOOL  ; Synthesis OK
H351.03 BOOL  ; Synthesis NG
H351.08 BOOL  ; OK WORKPIECE
H351.09 BOOL  ; Bearing insert having
H351.10 BOOL  ; Bearing press-fitting available (with guide operation)
H355.00 BOOL  ; 10ST_COMPLETE
H356.00 BOOL  ; LENGTH WORKPIECE
H356.02 BOOL  ; Synthesis OK
H356.03 BOOL  ; Synthesis NG
H356.04 BOOL  ; OVERALL LENGTH OK
H356.05 BOOL  ; OVERALL LENGTH NG
H356.06 BOOL  ; BEARING LENGTH OK
H356.07 BOOL  ; BEARING LENGTH NG
H356.08 BOOL  ; OK WORKPIECE
H356.09 BOOL  ; Bearing insert having
H356.10 BOOL  ; 10st operation disabled (valid at master)
H356.11 BOOL  ; Dimension measurement 0 master
H356.12 BOOL  ; Dimension measurement + NG master
H356.13 BOOL  ; Dimension measurement-NG master
H356.15 BOOL  ; Dimension measurement master work available
H357.00 BOOL  ; 0 MASTER SETTING COMPLETE
H357.02 BOOL  ; Upper limit check completed (functional check)
H357.03 BOOL  ; Lower limit check completed (functional check)
H361.00 BOOL  ; UNLOADING WORKPIECE
H361.01 BOOL  ; NO UNLOADING WORKPIECE
H361.02 BOOL  ; UNLOADING WORKPIECE Synthesis OK
H362.00 BOOL  ; WORKPIECE IN UNLOADING ROBOT CHUCK
H362.01 BOOL  ; NO WORKPIECE IN UNLOADING ROBOT CHUCK
H362.02 BOOL  ; UNLOADING ROBOT WORKPIECE Synthesis OK
H362.04 BOOL  ; INSURASION OK
H362.05 BOOL  ; INSURASION NG
H362.06 BOOL  ; Product number selection OK
H362.07 BOOL  ; Product number selection NG
H362.08 BOOL  ; SWING OK
H362.09 BOOL  ; SWING NG
H362.10 BOOL  ; RESISTANCE OK
H362.11 BOOL  ; RESISTANCE NG
H362.12 BOOL  ; IMPULSE OK
H362.13 BOOL  ; IMPULSE NG
H362.14 BOOL  ; OVERALL LENGTH OK
H362.15 BOOL  ; OVERALL LENGTH NG
H363.00 BOOL  ; UNLOADING TO LANE 1 (EXCHANGE CONTAINER)
H363.01 BOOL  ; UNLOADING TO LANE 2 (EXCHANGE CONTAINER)
H363.02 BOOL  ; UNLOADING TO LANE 1 (CONTAINER BEFOR EXCHANGE)
H363.03 BOOL  ; UNLOADING TO LANE 2 (CONTAINER BEFOR EXCHANGE)
H363.04 BOOL  ; Container exchange confirmation (Lane 1)
H363.05 BOOL  ; Container exchange confirmation (Lane 2)
H364.00 BOOL  ; Product number change 1 (Lane 1)
H364.01 BOOL  ; Product number change 1 (Lane 2)
H364.02 BOOL  ; Product number change 2 (Lane 1)
H364.03 BOOL  ; Product number change 2 (Lane 2)
H364.04 BOOL  ; Container exchange memory (Lane 1)(EXCHANGE CONTAINER)
H364.05 BOOL  ; Container exchange memory (Lane 2)(EXCHANGE CONTAINER)
H364.06 BOOL  ; Container exchange memory (Lane 1)(CONTAINER BEFOR EXCHANGE)
H364.07 BOOL  ; Container exchange memory (Lane 2)(CONTAINER BEFOR EXCHANGE)
H364.08 BOOL  ; Impropriety of stacking (Lane 1)
H364.09 BOOL  ; Impropriety of stacking (Lane 2)
H364.10 BOOL  ; Down confirmation when product number is switched (Lane 1)
H364.11 BOOL  ; Down confirmation when product number is switched (Lane 2)
H364.12 BOOL  ; STACKING CONTAINER DISCHARGE (LANE 1)
H364.13 BOOL  ; STACKING CONTAINER DISCHARGE (LANE 2)
H364.14 BOOL  ; DISCHARGING COMPLETE OF STACKING CONTAINER  (LANE 1)
H364.15 BOOL  ; DISCHARGING COMPLETE OF STACKING CONTAINER  (LANE 2)
H366.00 BOOL  ; BEARING PUSHER FORWARD MEMORY
H367.00 BOOL  ; UNLOADING LANE CONFIRMATION
H372.00 BOOL  ; DISCHARGING COMPLETE OF BEARING TRAY
H422 CHANNEL  ; Counter electrode resistance measurement OK (180 °)
H422.00 BOOL  ; NEXT RESISTANCE 1 OK
H422.01 BOOL  ; NEXT RESISTANCE 2 OK
H422.02 BOOL  ; NEXT RESISTANCE 3 OK
H422.03 BOOL  ; NEXT RESISTANCE 4 OK
H422.04 BOOL  ; NEXT RESISTANCE 4 OK
H422.05 BOOL  ; NEXT RESISTANCE 5 OK
H422.06 BOOL  ; NEXT RESISTANCE 6 OK
H422.07 BOOL  ; NEXT RESISTANCE 7 OK
H422.08 BOOL  ; NEXT RESISTANCE 8 OK
H423 CHANNEL  ; Counter electrode resistance measurement NG (180 °)
H423.00 BOOL  ; NEXT RESISTANCE 1 NG
H423.01 BOOL  ; NEXT RESISTANCE 2 NG
H423.02 BOOL  ; NEXT RESISTANCE 3 NG
H423.03 BOOL  ; NEXT RESISTANCE 4 NG
H423.04 BOOL  ; NEXT RESISTANCE 5 NG
H423.05 BOOL  ; NEXT RESISTANCE 6 NG
H423.06 BOOL  ; NEXT RESISTANCE 7 NG
H423.07 BOOL  ; NEXT RESISTANCE 8 NG
H423.08 BOOL  ; NEXT RESISTANCE 9 NG
H43 CHANNEL  ; palletizing shift of bearing supply robot
H43.09 BOOL  ; PALLETIZING COMPLETE
H460 CHANNEL  ; Memory of packing in a container of lane 1 (exchange container)
H460.00 BOOL  ; Memory 1 of packing in a container of lane 1 (exchange container)
H461.07 BOOL  ; Memory 24 of packing in a container of lane 1 (exchange container)
H462 CHANNEL  ; Memory of packing in a container of lane 1 (container befor exchange)
H462.00 BOOL  ; Memory 1 of packing in a container of lane 1 (container befor exchange)
H464 CHANNEL  ; Memory of packing in a container of lane 2 (exchange container)
H464.00 BOOL  ; Memory 1 of packing in a container of lane 2 (exchange container)
H465.07 BOOL  ; Memory 24 of packing in a container of lane 2 (exchange container)
H466 CHANNEL  ; Memory of packing in a container of lane 2 (container befor exchange)
H466.00 BOOL  ; Memory 1 of packing in a container of lane 2 (container befor exchange)
H470 CHANNEL  ; Memory of packing in a container of fraction workpiece
H470.00 BOOL  ; Memory 1 of packing in a container of fraction workpiece
H470.02 BOOL  ; Memory 3 of packing in a container of fraction workpiece
H470.04 BOOL  ; Memory 5 of packing in a container of fraction workpiece
H470.05 BOOL  ; Memory 6 of packing in a container of fraction workpiece
H470.08 BOOL  ; Memory 9 of packing in a container of fraction workpiece
H470.09 BOOL  ; Memory 10 of packing in a container of fraction workpiece
H470.11 BOOL  ; Memory 12 of packing in a container of fraction workpiece
H470.14 BOOL  ; Memory 15 of packing in a container of fraction workpiece
H471 CHANNEL  ; Memory of packing in a container of fraction workpiece
H471.01 BOOL  ; Memory 18 of packing in a container of fraction workpiece
H471.03 BOOL  ; Memory 20 of packing in a container of fraction workpiece
H471.05 BOOL  ; Memory 22 of packing in a container of fraction workpiece
H471.07 BOOL  ; Memory 24 of packing in a container of fraction workpiece
H510.02 BOOL  ; Re-input mode is being selected
H510.03 BOOL  ; Single operation is being selected
H510.04 BOOL  ; EL master work flow mode is being selected
H510.06 BOOL  ; Dimension master matching mode (LM) is being selected
H510.07 BOOL  ; Dimension Master Check Mode (LM) is being selected
H510.08 BOOL  ; Dimension master matching mode (S) is being selected
H510.09 BOOL  ; Dimension Master Check Mode (S) is being selected
H510.10 BOOL  ; Dimension Master Check Mode is being selected_Comprehensive
H6.00 BOOL  ; ボールと体格不一致
H6.01 BOOL  ; Body size switching operation_Payout completed
H8 CHANNEL  ; Master check step
H80.00 BOOL  ; Even number
T0001 BOOL  ; ID circuit start
T0002 BOOL  ; ID writing start
T0003 BOOL  ; Data reading start timing
T0004 BOOL  ; NG without ID1 storage data
T0005 BOOL  ; Timing of trigger
T0006 BOOL  ; Writing start timing
T0007 BOOL  ; Timing of trigger
T0009 BOOL  ; NO RESPONSE OF ID1
T0011 BOOL  ; ID circuit start
T0012 BOOL  ; ID writing start
T0013 BOOL  ; Data reading start timing
T0014 BOOL  ; NG without ID2 storage data
T0015 BOOL  ; Timing of trigger
T0016 BOOL  ; Writing start timing
T0017 BOOL  ; Timing of trigger
T0019 BOOL  ; NO RESPONSE OF ID2
T0021 BOOL  ; ID circuit start
T0022 BOOL  ; ID writing start
T0023 BOOL  ; Data reading start timing
T0024 BOOL  ; NG without ID3 storage data
T0025 BOOL  ; Timing of trigger
T0026 BOOL  ; Writing start timing
T0027 BOOL  ; Timing of trigger
T0029 BOOL  ; NO RESPONSE OF ID3
T0031 BOOL  ; ID circuit start
T0032 BOOL  ; ID writing start
T0033 BOOL  ; Data reading start timing
T0034 BOOL  ; NG without ID4 storage data
T0035 BOOL  ; Timing of trigger
T0036 BOOL  ; Writing start timing
T0037 BOOL  ; Timing of trigger
T0039 BOOL  ; NO RESPONSE OF ID4
T0095 BOOL  ; Program start delay
T0096 BOOL  ; Program start end
T0111 BOOL  ; BCD CHANGE TIME
T0115 BOOL  ; -
T0131 BOOL  ; INSULATION TEST END
T0132 BOOL  ; RESET TIME
T0133 BOOL  ; INSULATION TEST END
T0134 BOOL  ; Relay ON timer
T0135 BOOL  ; OK signal confirmation
T0136 BOOL  ; Relay switch time
T0137 BOOL  ; NUMBER OF TURNS CHECK TIMMING
T0138 BOOL  ; NUMBER OF TURNS CONFIRMATION TIMMING
T0140 BOOL  ; CONTACT PROBE IN RESISTANCE FORWARD END
T0141 BOOL  ; Measurement time
T0142 BOOL  ; RESISTANCE MEASUREMENT FINISH
T0143 BOOL  ; CONTACT PROBE IN RESISTANCE FORWARD END
T0144 BOOL  ; Resistance measurement TRIG
T0145 BOOL  ; CONTACT PROBE IN INPULSE FORWARD END
T0146 BOOL  ; Relay switch time (pair pole)
T0147 BOOL  ; Relay switch time (next pole)
T0148 BOOL  ; Page set time
T0149 BOOL  ; Page switch timer
T0155 BOOL  ; LENGTH MEASUREMENT FORWARD END
T0156 BOOL  ; Adjacent resistance measurement time
T0160 BOOL  ; WORKPIECE CLAMP IN LENGTH MEASURE DOWNWARD END
T0162 BOOL  ; UNLOADING ROBOT CHUCK CLAMP END
T0163 BOOL  ; UNLOADING ROBOT CHUCK UNCLAMP END
T0230 BOOL  ; Strobe start timing
T0240 BOOL  ; SIGNAL SWITCH WHEN STARTING
T0250 BOOL  ; POWER SUPPLY ON CHECK 1
T0251 BOOL  ; POWER SUPPLY ON CHECK 2
T0252 BOOL  ; MASTER SWITCH ON CHECK 1
T0253 BOOL  ; MASTER SWITCH ON CHECK 2
T0254 BOOL  ; One minute after power supply ON
T0255 BOOL  ; MASTER ON DERAY
T0257 BOOL  ; FULL DEFECTS
T0258 BOOL  ; WAITING FOR LOADING WORKPIECE
T0259 BOOL  ; IMPULSE ERROR
T0260 BOOL  ; LS FAULT 1
T0261 BOOL  ; LS FAULT 2
T0262 BOOL  ; LS FAULT 3
T0263 BOOL  ; LS FAULT 4
T0264 BOOL  ; LS FAULT 5
T0265 BOOL  ; LS FAULT 6
T0266 BOOL  ; LS FAULT 7
T0267 BOOL  ; LS FAULT 8
T0268 BOOL  ; LS FAULT 9
T0269 BOOL  ; LS FAULT 10
T0270 BOOL  ; LS FAULT 11
T0271 BOOL  ; LS FAULT 12
T0272 BOOL  ; LS FAULT 13
T0273 BOOL  ; LS FAULT 14
T0274 BOOL  ; LS FAULT 15
T0275 BOOL  ; LS FAULT 16
T0276 BOOL  ; LS FAULT 17
T0277 BOOL  ; LS FAULT 18
T0278 BOOL  ; LS FAULT 19
T0279 BOOL  ; LS FAULT 20
T0280 BOOL  ; LS FAULT 21
T0281 BOOL  ; LS FAULT 22
T0282 BOOL  ; LS FAULT 23
T0283 BOOL  ; LS FAULT 24
T0284 BOOL  ; LS FAULT 25
T0285 BOOL  ; LS FAULT 26
T0286 BOOL  ; LS FAULT 27
T0287 BOOL  ; LS FAULT 28
T0288 BOOL  ; LS FAULT 29
T0289 BOOL  ; LS FAULT 30
T0290 BOOL  ; LS FAULT 31
T0292 BOOL  ; LS FAULT 33
T0293 BOOL  ; LS FAULT 34
T0294 BOOL  ; LS FAULT 35
T0295 BOOL  ; LS FAULT 36
T0296 BOOL  ; Judgment invalidity timer
T0297 BOOL  ; Disconnection detection time of input 1
T0298 BOOL  ; WITHSTAND VOLTAGE TESTER FAULT
T0299 BOOL  ; The resistance bit is abnormal
T0300 BOOL  ; Sure PB effective time
T0301 BOOL  ; MASTER OFF
T0302 BOOL  ; AUTO / INDIV.
T0312 BOOL  ; CYCLE STOP
T0313 BOOL  ; 全作業終了運転スタート
T0316 BOOL  ; LS FAULT 59
T0317 BOOL  ; LS FAULT 60
T0320 BOOL  ; LS FAULT 37
T0321 BOOL  ; LS FAULT 38
T0322 BOOL  ; LS FAULT 39
T0323 BOOL  ; LS FAULT 40
T0324 BOOL  ; LS FAULT 41
T0325 BOOL  ; LS FAULT 42
T0326 BOOL  ; LS FAULT 43
T0327 BOOL  ; LS FAULT 44
T0328 BOOL  ; LS FAULT 45
T0329 BOOL  ; LS FAULT 46
T0330 BOOL  ; LS FAULT 47
T0331 BOOL  ; LS FAULT 48
T0332 BOOL  ; LS FAULT 49
T0333 BOOL  ; LS FAULT 50
T0334 BOOL  ; LS FAULT 51
T0335 BOOL  ; LS FAULT 52
T0336 BOOL  ; LS FAULT 53
T0337 BOOL  ; LS FAULT 54
T0338 BOOL  ; LS FAULT 55
T0339 BOOL  ; LS FAULT 56
T0340 BOOL  ; LS FAULT 57
T0341 BOOL  ; LS FAULT 58
T0342 BOOL  ; FULL CONTAINER (LANE 1)
T0343 BOOL  ; FULL CONTAINER (LANE 2)
T0344 BOOL  ; FULL BEARING TRAY
T0346 BOOL  ; CONTAINER DECREASING (LANE 1)
T0347 BOOL  ; CONTAINER DECREASING (LANE 2)
T0348 BOOL  ; BEARING TRAY DECREASING
T0350 BOOL  ; START CONFIRMATION
T0358 BOOL  ; Data clearness
T0361 BOOL  ; ROBOT MASTER ON
T0362 BOOL  ; FIXED POSITION RETURN
T0363 BOOL  ; FIXED POSITIONRETURN TIMMING
T0364 BOOL  ; Abnormal code reading timing
T0400 BOOL  ; AUTO RUNNING 30-SECOND PROGRESS
T0401 BOOL  ; LOADING CONVEYOR ON
T0402 BOOL  ; PALLET CHANGE TIMING OF ID RESET START SELECT
T0404 BOOL  ; DRIVING PREPARATION OFF CONFIRMATION
T0406 BOOL  ; ABS STARTING POINT SETTING
T0441 BOOL  ; X AXIS SERVO LOCK ON CONFIRMATION
T0500 BOOL  ; -
T0510 BOOL  ; RB_MSTR_ON_RUN_TR
T0511 BOOL  ; RB_HOME_POS_PB_TR
T0515 BOOL  ; STROBE_START_TIMING_TR
T0520 BOOL  ; SS_AUTO_TR
T0521 BOOL  ; SS_IND_TR
T0654 BOOL  ; Product number change confirmation
T0666 BOOL  ; SURE PB CONFIRMATION
T0800 BOOL  ; DERAY
T0900 BOOL  ; FLOW PRODUCT NUMBER CHANGE (WINDING No.1)
T0901 BOOL  ; FLOW PRODUCT NUMBER CHANGE (WINDING No.2)
T1100 BOOL  ; 01ST_CYCLE TIME OVER
T1101 BOOL  ; Condition waiting
T1110 BOOL  ; PALLET ON LOADING CONVEYOR
T1112 BOOL  ; WORKPIECE ON LOADING CONVEYOR
T1113 BOOL  ; NO WORKPIECE ON LOADING CONVEYOR
T1147 BOOL  ; Adjacent relay switching time (when displaying each individual _ waveform)
T1150 BOOL  ; 02ST_CY TIME OVER
T1151 BOOL  ; Condition waiting
T1159 BOOL  ; Workpiece chuck mistake check timing
T1161 BOOL  ; LOADER CHUCK UNCLAMP END
T1162 BOOL  ; LOADER CHUCK CLAMP END
T1200 BOOL  ; 03ST_CYCLE TIME OVER
T1250 BOOL  ; 04ST_CYCLE TIME OVER
T1252 BOOL  ; Distinction delay (thickness of core)
T1300 BOOL  ; 05ST_CYCLE TIME OVER
T1312 BOOL  ; insulation circuit check
T1350 BOOL  ; 06ST_CYCLE TIME OVER
T1360 BOOL  ; POSITIONING ARROW BACKWARD END
T1370 BOOL  ; High-speed workpiece rotation stability
T1371 BOOL  ; Swinging measurement time
T1372 BOOL  ; Middle-speed workpiece rotation stability
T1373 BOOL  ; Workpiece rotation stop confirmation
T1375 BOOL  ; POSITIONING RETRY TIMER
T1400 BOOL  ; 07ST_CYCLE TIME OVER
T1401 BOOL  ; Condition waiting
T1404 BOOL  ; RETRY TIMING
T1410 BOOL  ; WORKPIECE CLAMP IN RESISTANCE DOWNWARD END
T1411 BOOL  ; CONTACT PROBE IN RESISTANCE BACKWARD END
T1450 BOOL  ; 08ST_CYCLE TIME OVER
T1451 BOOL  ; Condition waiting
T1452 BOOL  ; Master Check Delay Time Over
T1456 BOOL  ; RETRY TIMING (IMPULSE)
T1460 BOOL  ; WORKPIECE CLAMP IN INPULSE DOWNWARD END
T1461 BOOL  ; CONTACT PROBE IN INPULSE BACKWARD END
T1470 BOOL  ; Relay switch timing
T1471 BOOL  ; Relay switch timing
T1500 BOOL  ; 09ST_CYCLE TIME OVER
T1501 BOOL  ; Condition waiting
T1502 BOOL  ; INSERT TIME
T1511 BOOL  ; BEARING INSERT (HIGH PRESSURE) OFF
T1512 BOOL  ; BEARING CONFIRMATION
T1513 BOOL  ; NO BEARING
T1514 BOOL  ; BEARING BEFORE INSERT
T1515 BOOL  ; NO BEARING BEFORE INSERT
T1517 BOOL  ; BEARING INSERT (HIGH SPEED) BACKWARD TIME
T1518 BOOL  ; Bearing press-fit work presser rising end
T1519 BOOL  ; Bearing guide forward end timer
T1550 BOOL  ; 10ST_CYCLE TIME OVER
T1551 BOOL  ; -
T1552 BOOL  ; CHECK TIME
T1570 BOOL  ; ZERO RESET TIMING
T1600 BOOL  ; 11ST_CYCLE TIME OVER
T1605 BOOL  ; Condition waiting
T1610 BOOL  ; CONTAINER CONFIRMATION
T1611 BOOL  ; NO CONTAINER
T1612 BOOL  ; ROBOT DISCHARGE WAITING
T1613 BOOL  ; Compulsion retreat signal
T1650 BOOL  ; 12ST_CYCLE TIME OVER
T1652 BOOL  ; BEARING DOWNWARD DERAY
T1660 BOOL  ; -
T1661 BOOL  ; FULL BEARING OFF
T1662 BOOL  ; BEARING TRANSFER CARRIER FORWARD END TIME
T1663 BOOL  ; BEARING TRANSFER DOWNWARD END TIME
T1664 BOOL  ; BEARING PUSHER BACKWARD TIME
T1665 BOOL  ; BEARING PUSHER FORWARD MEMORY TIME
T1667 BOOL  ; BEARING TRANSFER UPWARD END CONFIRMATION
T1670 BOOL  ; BEARING TRANSFER DOWNWARD TIME
T1671 BOOL  ; BEARING TRANSFER DOWNWARD OFF
T1700 BOOL  ; 13ST_CYCLE TIME OVER
T1702 BOOL  ; Condition waiting
T1703 BOOL  ; CONVEYOR ROTATE
T1710 BOOL  ; LOADING BEARING TRAY
T1711 BOOL  ; NO LOADING BEARING TRAY
T1712 BOOL  ; BEARING TRAY BEFOR EXCHANGE
T1713 BOOL  ; NO BEARING TRAY BEFOR EXCHANGE
T1714 BOOL  ; EXCHANGE BEARING TRAY
T1715 BOOL  ; NO EXCHANGE BEARING TRAY
T1716 BOOL  ; PASSING BEARING TRAY ON
T1717 BOOL  ; PASSING BEARING TRAY OFF
T1718 BOOL  ; PASSING UNLOADING BEARING TRAY ON
T1719 BOOL  ; PASSING UNLOADING BEARING TRAY OFF
T1750 BOOL  ; 14ST_CYCLE TIME OVER
T1760 BOOL  ; WORKPIECE ON DEFECT DISCHARGING CONVEYOR
T1761 BOOL  ; NO WORKPIECE ON DEFECT DISCHARGING CONVEYOR
T1762 BOOL  ; FULL WORKPIECES ON DEFECT DISCHARGING CONVEYOR IS TURNED ON
T1763 BOOL  ; FULL WORKPIECES ON DEFECT DISCHARGING CONVEYOR IS TURNED OFF
T1764 BOOL  ; DEFECT DISCHARGING CONVEYOR PAEKING POSITION IS TURNED ON
T1765 BOOL  ; DEFECT DISCHARGING CONVEYOR PAEKING POSITION IS TURNED OFF
T1800 BOOL  ; 15ST_CYCLE TIME OVER
T1802 BOOL  ; Condition waiting
T1803 BOOL  ; LOADING CONVEYOR
T1810 BOOL  ; LOADING CONTAINER
T1811 BOOL  ; NO LOADING CONTAINER
T1812 BOOL  ; CONTAINER BEFOR PALLETIZING
T1813 BOOL  ; NO CONTAINER BEFOR PALLETIZING
T1814 BOOL  ; PALLETIZING CONTAINER
T1815 BOOL  ; NO PALLETIZING CONTAINER
T1816 BOOL  ; PALLETIZING CONTAINER UPPER SECTION
T1817 BOOL  ; NO PALLETIZING CONTAINER UPPER SECTION
T1818 BOOL  ; CONTAINER DECREASING
T1819 BOOL  ; NO LOADING CONTAINER
T1821 BOOL  ; NO CONTAINER BEFOR PALLETIZING
T1850 BOOL  ; 16ST_CYCLE TIME OVER
T1852 BOOL  ; Condition waiting
T1860 BOOL  ; CONTAINER BEFOR EXCHANGE
T1861 BOOL  ; NO CONTAINER BEFOR EXCHANGE
T1862 BOOL  ; EXCHANGE CONTAINER
T1863 BOOL  ; NO EXCHANGE CONTAINER
T1864 BOOL  ; CONFIRMATION ON (PASSING EXCHANGE CONTAINER)
T1865 BOOL  ; CONFIRMATION ON (PASSING EXCHANGE CONTAINER)
T1900 BOOL  ; 17ST_CYCLE TIME OVER
T1901 BOOL  ; Forced ending
T1902 BOOL  ; Condition waiting
T1903 BOOL  ; UNLOADING CONVEYOR 1&2
T1904 BOOL  ; DOWNWARD END (At the switch of the product number)
T1906 BOOL  ; Container sending time
T1910 BOOL  ; STACKING CONTAINER
T1911 BOOL  ; NO STACKING CONTAINER
T1912 BOOL  ; CONFIRMATION ON (STACKING CONTAINER UPPER SECTION)
T1913 BOOL  ; CONFIRMATION ON (STACKING CONTAINER UPPER SECTION)
T1914 BOOL  ; CONFIRMATION ON (FULL CONTAINERS ON UNLOADING CONVEYOR)
T1915 BOOL  ; CONFIRMATION ON (FULL CONTAINERS ON UNLOADING CONVEYOR)
T1916 BOOL  ; CONFIRMATION ON (UNLOADING CONTAINERS)
T1917 BOOL  ; CONFIRMATION ON (UNLOADING CONTAINERS)
T1950 BOOL  ; 18ST_CYCLE TIME OVER
T1952 BOOL  ; Condition waiting
T1953 BOOL  ; LOADING CONVEYOR
T1960 BOOL  ; LOADING CONTAINER
T1961 BOOL  ; NO LOADING CONTAINER
T1962 BOOL  ; CONTAINER BEFOR PALLETIZING
T1963 BOOL  ; NO CONTAINER BEFOR PALLETIZING
T1964 BOOL  ; PALLETIZING CONTAINER
T1965 BOOL  ; NO PALLETIZING CONTAINER
T1966 BOOL  ; PALLETIZING CONTAINER UPPER SECTION
T1967 BOOL  ; NO PALLETIZING CONTAINER UPPER SECTION
T1968 BOOL  ; CONTAINER DECREASING
T1969 BOOL  ; NO LOADING CONTAINER
T1971 BOOL  ; NO CONTAINER BEFOR PALLETIZING
T2000 BOOL  ; 19ST_CYCLE TIME OVER
T2002 BOOL  ; Condition waiting
T2010 BOOL  ; CONTAINER BEFOR EXCHANGE
T2011 BOOL  ; NO CONTAINER BEFOR EXCHANGE
T2012 BOOL  ; EXCHANGE CONTAINER
T2013 BOOL  ; NO EXCHANGE CONTAINER
T2014 BOOL  ; CONFIRMATION ON (PASSING EXCHANGE CONTAINER)
T2015 BOOL  ; CONFIRMATION ON (PASSING EXCHANGE CONTAINER)
T2050 BOOL  ; 20ST_CYCLE TIME OVER
T2051 BOOL  ; Forced ending
T2052 BOOL  ; Condition waiting
T2053 BOOL  ; UNLOADING CONVEYOR 1&2
T2054 BOOL  ; DOWNWARD END (At the switch of the product number)
T2056 BOOL  ; Container sending time
T2060 BOOL  ; STACKING CONTAINER
T2061 BOOL  ; NO STACKING CONTAINER
T2062 BOOL  ; CONFIRMATION ON (STACKING CONTAINER UPPER SECTION)
T2063 BOOL  ; CONFIRMATION ON (STACKING CONTAINER UPPER SECTION)
T2064 BOOL  ; CONFIRMATION ON (FULL CONTAINERS ON UNLOADING CONVEYOR)
T2065 BOOL  ; CONFIRMATION ON (FULL CONTAINERS ON UNLOADING CONVEYOR)
T2066 BOOL  ; CONFIRMATION ON (UNLOADING CONTAINERS)
T2067 BOOL  ; CONFIRMATION ON (UNLOADING CONTAINERS)
T2070 BOOL  ; STACKING LIFTER UPWARD END
T3010 BOOL  ; LANGUAGE CHANGE
W0.00 BOOL  ; MASTER SWITCH ON
W0.01 BOOL  ; AUTO START
W0.02 BOOL  ; CYCLE STOP
W0.03 BOOL  ; ALL HOME POSITION RETURN
W0.04 BOOL  ; OPERATION AUTO/IND SELECT
W0.06 BOOL  ; OK_PBon
W0.08 BOOL  ; YES_PBon
W0.09 BOOL  ; NO_PBon
W0.12 BOOL  ; FAULT RESET
W0.13 BOOL  ; ALARM RESET
W0.15 BOOL  ; FAULT DISPLAY FLICKER
W104.00 BOOL  ; NUMBER OF TURNS CHECK RELAY ON
W104.04 BOOL  ; NUMBER OF TURNS CHECK START PL
W105.00 BOOL  ; NUMBER OF TURNS CHECK COMPLETE
W10.01 BOOL  ; ROBOR FIXED POSITION
W10.02 BOOL  ; ROBOT READY
W10.03 BOOL  ; BEARING SUPPLY ROBOT FIXED POSITION
W10.04 BOOL  ; CONDITION OF MASTER ON
W10.05 BOOL  ; CONDITION OF AUTO START
W10.13 BOOL  ; Staking Not Use (Line 1)
W11.00 BOOL  ; ID operation invalidity
W11.01 BOOL  ; Dimension Master Check Mode (LM) Selection PB
W11.02 BOOL  ; LANE 1 CONFIRMATION THE OPERATION
W11.03 BOOL  ; LANE 2 CONFIRMATION THE OPERATION
W11.11 BOOL  ; by Nanang For memory shifting
W120.00 BOOL  ; FUSE GOOD
W120.01 BOOL  ; THERMAL GOOD
W120.02 BOOL  ; SAFETY GUARD CLOSE
W120.03 BOOL  ; PC OK
W120.05 BOOL  ; EXCHANGE CONTAINER
W120.06 BOOL  ; EXCHANGE CONTAINER
W120.07 BOOL  ; CONTAINER CONFIRMATION
W120.08 BOOL  ; CONTAINER BEFOR EXCHANGE
W120.09 BOOL  ; CONTAINER BEFOR EXCHANGE
W121.00 BOOL  ; ALL HOME POSITION
W121.01 BOOL  ; WORKPIECE CONFITION
W121.02 BOOL  ; TEACHING OFF
W121.03 BOOL  ; ROBOT FIXED POSITION
W121.04 BOOL  ; WITH.VOL.READY
W121.05 BOOL  ; MASTER SETTING COMPLETE
W121.07 BOOL  ; RESISTANCE MEASURE READY
W121.08 BOOL  ; INPULSE TESTER READY
W121.09 BOOL  ; BEARING SUPPLY ROBOT READY
W121.10 BOOL  ; FORMER PROCESS CONVEYOR ON
W122.00 BOOL  ; 01ST_HOME POSITION
W122.01 BOOL  ; 02ST_HOME POSITION
W122.02 BOOL  ; 03ST_HOME POSITION
W122.03 BOOL  ; 04ST_HOME POSITION
W122.04 BOOL  ; 05ST_HOME POSITION
W122.05 BOOL  ; 06ST_HOME POSITION
W122.06 BOOL  ; 7ST_HOME POSITION
W122.07 BOOL  ; 8ST_HOME POSITION
W122.08 BOOL  ; 9ST_HOME POSITION
W122.09 BOOL  ; 10ST_HOME POSITION
W123.00 BOOL  ; 11ST_HOME POSITION
W123.01 BOOL  ; 12ST_HOME POSITION
W123.02 BOOL  ; 13ST_HOME POSITION
W123.03 BOOL  ; 14ST_HOME POSITION
W123.04 BOOL  ; 15ST_HOME POSITION
W123.05 BOOL  ; 16ST_HOME POSITION
W123.06 BOOL  ; 17ST_HOME POSITION
W123.07 BOOL  ; 18ST_HOME POSITION
W123.08 BOOL  ; 19ST_HOME POSITION
W123.09 BOOL  ; 20ST_HOME POSITION
W125.00 BOOL  ; INSULATION TEST OK
W125.01 BOOL  ; SWING MEASUREMENT OK
W125.02 BOOL  ; RESISTANCE MEASUREMENT OK
W125.03 BOOL  ; Product number distinction OK (180)
W125.04 BOOL  ; IMPULSE MEASUREMENT OK
W125.05 BOOL  ; LENGTH MEASUREMENT OK
W125.06 BOOL  ; INSULATION TEST NG
W125.07 BOOL  ; SWING MEASUREMENT NG
W125.08 BOOL  ; RESISTANCE MEASUREMENT NG
W125.09 BOOL  ; Product number distinction NG (180)
W125.10 BOOL  ; IMPULSE MEASUREMENT NG
W125.11 BOOL  ; LENGTH MEASUREMENT NG
W126.00 BOOL  ; BEARING INSERT MEASUREMENT OK
W126.06 BOOL  ; BEARING INSERT MEASUREMENT NG
W12.00 BOOL  ; ID operation invalidity
W12.01 BOOL  ; Dimension Master Check Mode (LM) selected PL
W12.02 BOOL  ; LANE 1 CONFIRMATION THE OPERATION
W12.03 BOOL  ; LANE 2 CONFIRMATION THE OPERATION
W138.00 BOOL  ; MASTER ON PERMISSION
W138.01 BOOL  ; SAFETY DOOR OPEN OK(FROM PLC)
W138.02 BOOL  ; CONVEYOR ON PERMISSION
W138.03 BOOL  ; CONVEYOR ECO RUNNING 1
W138.04 BOOL  ; MASTER SWITCH ON
W138.05 BOOL  ; CONVEYOR SWITCH ON
W138.06 BOOL  ; CONVEYOR ECO RUNNING 2
W138.07 BOOL  ; ROBOT STOP FROM PLC(AT OFF)
W138.14 BOOL  ; ROBOT MASTER ON MC-B
W138.15 BOOL  ; OTHER MASTER ON MC-C
W139.00 BOOL  ; FUSE GOOD
W139.01 BOOL  ; THERMAL RELAY GOOD
W139.02 BOOL  ; SAFETY CONFIRM 1-1(SAFETY DOOR SWITCH 1 CLOSE WHEN TEACHING ROBOT)
W139.03 BOOL  ; EX. HANDLE CONFIRMATION
W139.04 BOOL  ; SAFETY CONFIRM 2-1(SAFETY DOOR SWITCH 1 OPEN WHEN TEACHING ROBOT)
W139.05 BOOL  ; AIR CONFIRMATION
W139.06 BOOL  ; CONVEYOR THERMAL RELAY GOOD
W139.07 BOOL  ; MASTER ON CONFIRM
W139.08 BOOL  ; CONVEYOR ON CONFIRM
W139.09 BOOL  ; SAFETY CONFIRM 1-2(SAFETY DOOR SWITCH 2 CLOSE WHEN TEACHING ROBOT)
W139.10 BOOL  ; SAFETY CONFIRM 2-2(SAFETY DOOR SWITCH 2 OPEN WHEN TEACHING ROBOT)
W139.11 BOOL  ; SAFTY CONFIRM INVALID(KEY SWITCH TEACH ON)
W139.12 BOOL  ; EMERGENCY STOP PUSH BUTTON SWITCH OFF
W139.13 BOOL  ; SAFTY CONFIRM INVALID PL
W139.14 BOOL  ; MASTER ON COND.(EXT. A SAFEGUARD)
W139.15 BOOL  ; OPERATION PANEL SURE PUSH BUTTON SWITCH
W13.00 BOOL  ; PB_M/C SIGNL OPRATE
W140.00 BOOL  ; SET VALUE CHANGE INTERLOCK 1
W140.01 BOOL  ; SET VALUE CHANGE INTERLOCK 2
W142.00 BOOL  ; WORKPIECE NUMBER SELECTION +
W142.01 BOOL  ; WORKPIECE NUMBER SELECTION -
W142.02 BOOL  ; WORKPIECE NUMBER DATA REGISTRATION
W143.02 BOOL  ; WORKPIECE NUMBER DATA REGISTRATION
W150 CHANNEL  ; HEAD FAULT INDICATION CH
W150.00 BOOL  ; EMERG STOP:LOADING C/V PALLET SHIFT LS FAULT
W150.01 BOOL  ; EMERG STOP:LOADING C/V PALLET DISCHARGE LS FAULT
W150.02 BOOL  ; EMERG STOP:LOADER FORWARD-BACKWARD LS FAULT
W150.03 BOOL  ; EMERG STOP:LOADER UPWARD-DOWNWARD LS FAULT
W150.04 BOOL  ; EMERG STOP:LOADER CHUCK TURN-RETURN LS FAULT
W150.05 BOOL  ; EMERG STOP:LOADER CHUCK CLAMP-UNCLAMP LS FAULT
W150.06 BOOL  ; EMERG STOP:SUB TRANSFER CARRIER LIFTER LS FAULT
W150.07 BOOL  ; EMERG STOP:WORKPIECE PUSHER LS FAULT
W150.08 BOOL  ; EMERG STOP:TRANSFER CARRIER LS FAULT
W150.09 BOOL  ; EMERG STOP:WORKPIECE LIFTER LS FAULT
W150.10 BOOL  ; EMERG STOP:POSITIONING ARROW LS FAULT
W150.11 BOOL  ; EMERG STOP:RESISTANCE WORKPIECE CLAMP LS FAULT
W150.12 BOOL  ; EMERG STOP:RESISTANCE PROBE LS FAULT
W150.13 BOOL  ; EMERG STOP:IMPULSE WORKPIECE CLAMP LS FAULT
W150.14 BOOL  ; EMERG STOP:IMPULSE PROBE LS FAULT
W150.15 BOOL  ; EMERG STOP:LENGTH MEASUREMENT LS FAULT
W151.00 BOOL  ; EMERG STOP:UNLOADING ROBOT CHUCK LS FAULT
W151.01 BOOL  ; EMERG STOP:BEARING INSERT (HIGH PRESS) LS FAULT
W151.02 BOOL  ; EMERG STOP:BEARING INSERT (HIGH SPEED) LS FAULT
W151.03 BOOL  ; EMERG STOP:BEARING SHUTTER LS FAULT
W151.04 BOOL  ; EMERG STOP:BEARING GUIDE LS FAULT
W151.05 BOOL  ; EMERG STOP:BEARING ESCAPE LS FAULT
W151.06 BOOL  ; EMERG STOP:BEARING TRANSFER LS FAULT
W151.07 BOOL  ; EMERG STOP:BEARING PUSHER LS FAULT
W151.08 BOOL  ; EMERG STOP:BEARING TRANSFER CARRIER LS FAULT
W151.09 BOOL  ; EMERG STOP:BEARING HANGER FORWARD-BACKWARD LS FAULT
W151.10 BOOL  ; EMERG STOP:BEARING HANGER UPWARD-DOWNWARD LS FAULT
W151.11 BOOL  ; EMERG STOP:BEARING TRAY HOME POSITIONING LS FAULT
W151.12 BOOL  ; EMERG STOP:BEARING TRAY EXCHANGE LS FAULT
W151.13 BOOL  ; EMERG STOP:BEARING TRAY STOPPER LS FAULT
W151.14 BOOL  ; EMERG STOP:BEARING TRAY ESCAPE LS FAULT
W152.00 BOOL  ; EMERG STOP:LANE 1 POSITIONING 1 LS FAULT
W152.01 BOOL  ; EMERG STOP:LANE 1 POSITIONING 2 LS FAULT
W152.02 BOOL  ; EMERG STOP:LANE 1 LIFTER LS FAULT
W152.03 BOOL  ; EMERG STOP:LANE 1 DROP GUARD LS FAULT
W152.04 BOOL  ; EMERG STOP:LANE 1 PALLETIZING STOPPER LS FAULT
W152.05 BOOL  ; EMERG STOP:LANE 1 STOPPER BEFOR PALLETIZING LS FAULT
W152.06 BOOL  ; EMERG STOP:LANE 1 ESCAPE BEFOR PALLETIZING LS FAULT
W152.07 BOOL  ; EMERG STOP:LANE 1 PALLETIZING LIFTER LS FAULT
W152.08 BOOL  ; EMERG STOP:LANE 1 PALLETIZING HOOK LS FAULT
W152.09 BOOL  ; EMERG STOP:LANE 1 STACKING LIFTER LS FAULT
W152.10 BOOL  ; EMERG STOP:LANE 1 STACKING HOOK LS FAULT
W152.11 BOOL  ; EMERG STOP:LANE 1 STACKING STOPPER LS FAULT
W152.12 BOOL  ; EMERG STOP:LANE 1 UNLOADING STOPPER LS FAULT
W152.13 BOOL  ; EMERG STOP:LANE 1 UNLOADING ESCAPE LS FAULT
W152.14 BOOL  ; EMERG STOP:LANE 2 POSITIONING 1 LS FAULT
W152.15 BOOL  ; EMERG STOP:LANE 2 POSITIONING 2 LS FAULT
W153.00 BOOL  ; EMERG STOP:LANE 2 LIFTER LS FAULT
W153.01 BOOL  ; EMERG STOP:LANE 2 DROP GUARD LS FAULT
W153.02 BOOL  ; EMERG STOP:LANE 2 PALLETIZING STOPPER LS FAULT
W153.03 BOOL  ; EMERG STOP:LANE 2 STOPPER BEFOR PALLETIZING LS FAULT
W153.04 BOOL  ; EMERG STOP:LANE 2 ESCAPE BEFOR PALLETIZING LS FAULT
W153.05 BOOL  ; EMERG STOP:LANE 2 PALLETIZING LIFTER LS FAULT
W153.06 BOOL  ; EMERG STOP:LANE 2 PALLETIZING HOOK LS FAULT
W153.07 BOOL  ; EMERG STOP:LANE 2 STACKING LIFTER LS FAULT
W153.08 BOOL  ; EMERG STOP:LANE 2 STACKING HOOK LS FAULT
W153.09 BOOL  ; EMERG STOP:LANE 2 STACKING STOPPER LS FAULT
W153.10 BOOL  ; EMERG STOP:LANE 2 UNLOADING STOPPER LS FAULT
W153.11 BOOL  ; EMERG STOP:LANE 2 UNLOADING ESCAPE LS FAULT
W154.01 BOOL  ; EMERG STOP:AD UNIT FAULT
W154.02 BOOL  ; EMERG STOP:HIGH-SPEED COUNTER UNIT OF No.20 FAULT
W154.03 BOOL  ; EMERG STOP:HIGH-SPEED COUNTER UNIT OF No.24 FAULT
W154.12 BOOL  ; EMERG STOP:TRAY EXCHANGE INVERTER FAULT
W154.13 BOOL  ; EMERG STOP:BEARING SUPPRY ROBOT FAULT
W154.14 BOOL  ; EMERG STOP:DEFECTS DISCHARGING INVERTER FAULT
W154.15 BOOL  ; EMERG STOP:UNLOADING ROBOT FAULT
W155.00 BOOL  ; EMERG STOP:FUSE TRIP
W155.01 BOOL  ; EMERG STOP:MOTOR OVER-LOAD
W155.03 BOOL  ; EMERG STOP:AIR DECREASING
W155.04 BOOL  ; EMERG STOP:PC FAULT
W155.05 BOOL  ; EMERG STOP:COMPOBUS/S OUT COMMUNICATION OF No.0 FAULT
W155.06 BOOL  ; EMERG STOP:COMPOBUS/S IN COMMUNICATION OF No.0 FAULT
W155.07 BOOL  ; EMERG STOP:COMPOBUS/S OUT COMMUNICATION OF No.2 FAULT
W155.08 BOOL  ; EMERG STOP:COMPOBUS/S IN COMMUNICATION OF No.2 FAULT
W155.09 BOOL  ; EMERG STOP:COMPOBUS/S OUT COMMUNICATION OF No.4 FAULT
W155.10 BOOL  ; EMERG STOP:COMPOBUS/S IN COMMUNICATION OF No.4 FAULT
W155.11 BOOL  ; EMERG STOP:COMPOBUS/S OUT COMMUNICATION OF No.8 FAULT
W155.12 BOOL  ; EMERG STOP:COMPOBUS/S IN COMMUNICATION OF No.8 FAULT
